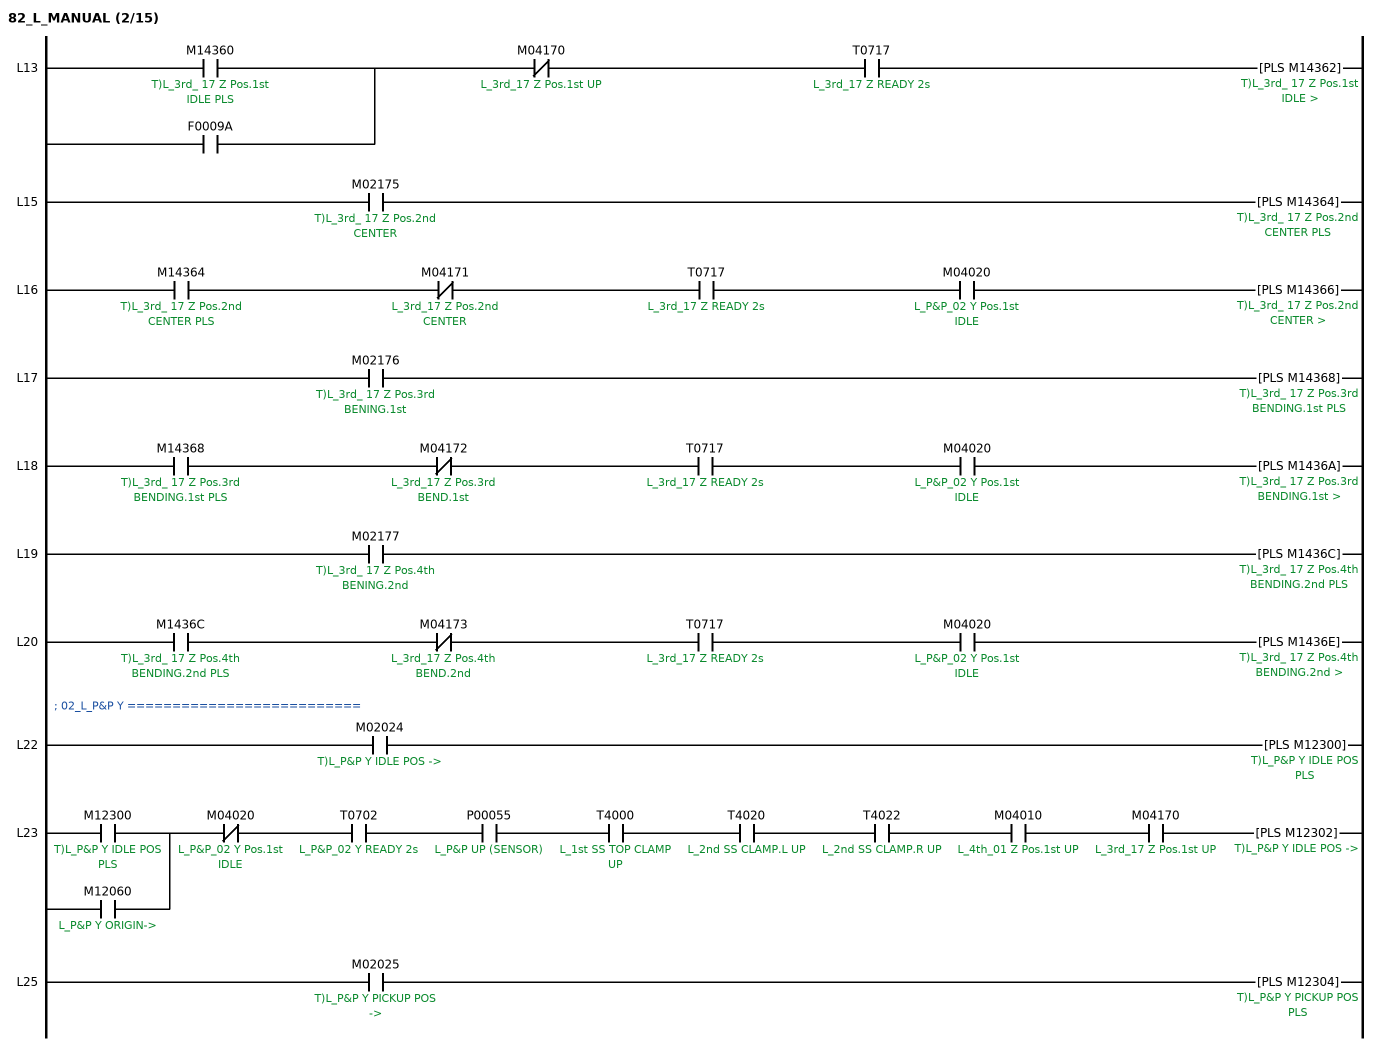
[picture p336: 82_L_MANUAL rungs L13-L25]
; L13
LOAD      M14360	// T)L_3rd_ 17 Z Pos.1st IDLE PLS
OR        F0009A
AND NOT   M04170	// L_3rd_17 Z Pos.1st UP
AND       T0717	// L_3rd_17 Z READY 2s
OUTP      M14362	// T)L_3rd_ 17 Z Pos.1st IDLE >
; L15
LOAD      M02175	// T)L_3rd_ 17 Z Pos.2nd CENTER
OUTP      M14364	// T)L_3rd_ 17 Z Pos.2nd CENTER PLS
; L16
LOAD      M14364	// T)L_3rd_ 17 Z Pos.2nd CENTER PLS
AND NOT   M04171	// L_3rd_17 Z Pos.2nd CENTER
AND       T0717	// L_3rd_17 Z READY 2s
AND       M04020	// L_P&P_02 Y Pos.1st IDLE
OUTP      M14366	// T)L_3rd_ 17 Z Pos.2nd CENTER >
; L17
LOAD      M02176	// T)L_3rd_ 17 Z Pos.3rd BENING.1st
OUTP      M14368	// T)L_3rd_ 17 Z Pos.3rd BENDING.1st PLS
; L18
LOAD      M14368	// T)L_3rd_ 17 Z Pos.3rd BENDING.1st PLS
AND NOT   M04172	// L_3rd_17 Z Pos.3rd BEND.1st
AND       T0717	// L_3rd_17 Z READY 2s
AND       M04020	// L_P&P_02 Y Pos.1st IDLE
OUTP      M1436A	// T)L_3rd_ 17 Z Pos.3rd BENDING.1st >
; L19
LOAD      M02177	// T)L_3rd_ 17 Z Pos.4th BENING.2nd
OUTP      M1436C	// T)L_3rd_ 17 Z Pos.4th BENDING.2nd PLS
; L20
LOAD      M1436C	// T)L_3rd_ 17 Z Pos.4th BENDING.2nd PLS
AND NOT   M04173	// L_3rd_17 Z Pos.4th BEND.2nd
AND       T0717	// L_3rd_17 Z READY 2s
AND       M04020	// L_P&P_02 Y Pos.1st IDLE
OUTP      M1436E	// T)L_3rd_ 17 Z Pos.4th BENDING.2nd >
// 02_L_P&P Y ==========================
; L22
LOAD      M02024	// T)L_P&P Y IDLE POS ->
OUTP      M12300	// T)L_P&P Y IDLE POS PLS
; L23
LOAD      M12300	// T)L_P&P Y IDLE POS PLS
OR        M12060	// L_P&P Y ORIGIN->
AND NOT   M04020	// L_P&P_02 Y Pos.1st IDLE
AND       T0702	// L_P&P_02 Y READY 2s
AND       P00055	// L_P&P UP (SENSOR)
AND       T4000	// L_1st SS TOP CLAMP    UP
AND       T4020	// L_2nd SS CLAMP.L UP
AND       T4022	// L_2nd SS CLAMP.R UP
AND       M04010	// L_4th_01 Z Pos.1st UP
AND       M04170	// L_3rd_17 Z Pos.1st UP
OUTP      M12302	// T)L_P&P Y IDLE POS ->
; L25
LOAD      M02025	// T)L_P&P Y PICKUP POS ->
OUTP      M12304	// T)L_P&P Y PICKUP POS PLS

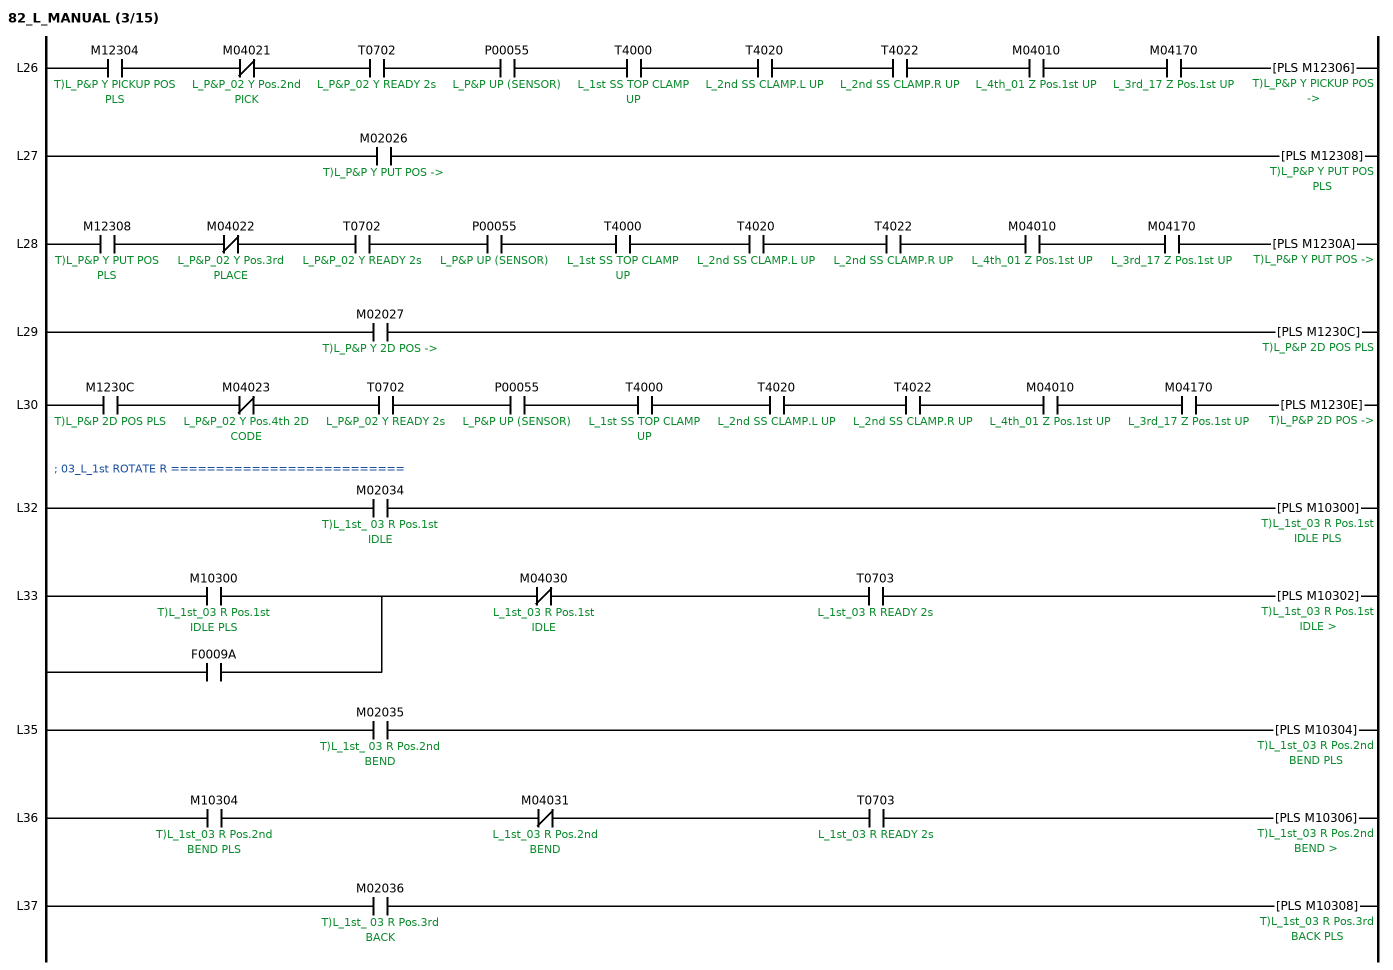
; L26
LOAD      M12304	// T)L_P&P Y PICKUP POS PLS
AND NOT   M04021	// L_P&P_02 Y Pos.2nd PICK
AND       T0702	// L_P&P_02 Y READY 2s
AND       P00055	// L_P&P UP (SENSOR)
AND       T4000	// L_1st SS TOP CLAMP    UP
AND       T4020	// L_2nd SS CLAMP.L UP
AND       T4022	// L_2nd SS CLAMP.R UP
AND       M04010	// L_4th_01 Z Pos.1st UP
AND       M04170	// L_3rd_17 Z Pos.1st UP
OUTP      M12306	// T)L_P&P Y PICKUP POS ->
; L27
LOAD      M02026	// T)L_P&P Y PUT POS ->
OUTP      M12308	// T)L_P&P Y PUT POS PLS
; L28
LOAD      M12308	// T)L_P&P Y PUT POS PLS
AND NOT   M04022	// L_P&P_02 Y Pos.3rd PLACE
AND       T0702	// L_P&P_02 Y READY 2s
AND       P00055	// L_P&P UP (SENSOR)
AND       T4000	// L_1st SS TOP CLAMP    UP
AND       T4020	// L_2nd SS CLAMP.L UP
AND       T4022	// L_2nd SS CLAMP.R UP
AND       M04010	// L_4th_01 Z Pos.1st UP
AND       M04170	// L_3rd_17 Z Pos.1st UP
OUTP      M1230A	// T)L_P&P Y PUT POS ->
; L29
LOAD      M02027	// T)L_P&P Y 2D POS ->
OUTP      M1230C	// T)L_P&P 2D POS PLS
; L30
LOAD      M1230C	// T)L_P&P 2D POS PLS
AND NOT   M04023	// L_P&P_02 Y Pos.4th 2D CODE
AND       T0702	// L_P&P_02 Y READY 2s
AND       P00055	// L_P&P UP (SENSOR)
AND       T4000	// L_1st SS TOP CLAMP    UP
AND       T4020	// L_2nd SS CLAMP.L UP
AND       T4022	// L_2nd SS CLAMP.R UP
AND       M04010	// L_4th_01 Z Pos.1st UP
AND       M04170	// L_3rd_17 Z Pos.1st UP
OUTP      M1230E	// T)L_P&P 2D POS ->
// 03_L_1st ROTATE R ==========================
; L32
LOAD      M02034	// T)L_1st_ 03 R Pos.1st IDLE
OUTP      M10300	// T)L_1st_03 R Pos.1st IDLE PLS
; L33
LOAD      M10300	// T)L_1st_03 R Pos.1st IDLE PLS
OR        F0009A
AND NOT   M04030	// L_1st_03 R Pos.1st IDLE
AND       T0703	// L_1st_03 R READY 2s
OUTP      M10302	// T)L_1st_03 R Pos.1st IDLE >
; L35
LOAD      M02035	// T)L_1st_ 03 R Pos.2nd BEND
OUTP      M10304	// T)L_1st_03 R Pos.2nd BEND PLS
; L36
LOAD      M10304	// T)L_1st_03 R Pos.2nd BEND PLS
AND NOT   M04031	// L_1st_03 R Pos.2nd BEND
AND       T0703	// L_1st_03 R READY 2s
OUTP      M10306	// T)L_1st_03 R Pos.2nd BEND >
; L37
LOAD      M02036	// T)L_1st_ 03 R Pos.3rd BACK
OUTP      M10308	// T)L_1st_03 R Pos.3rd BACK PLS

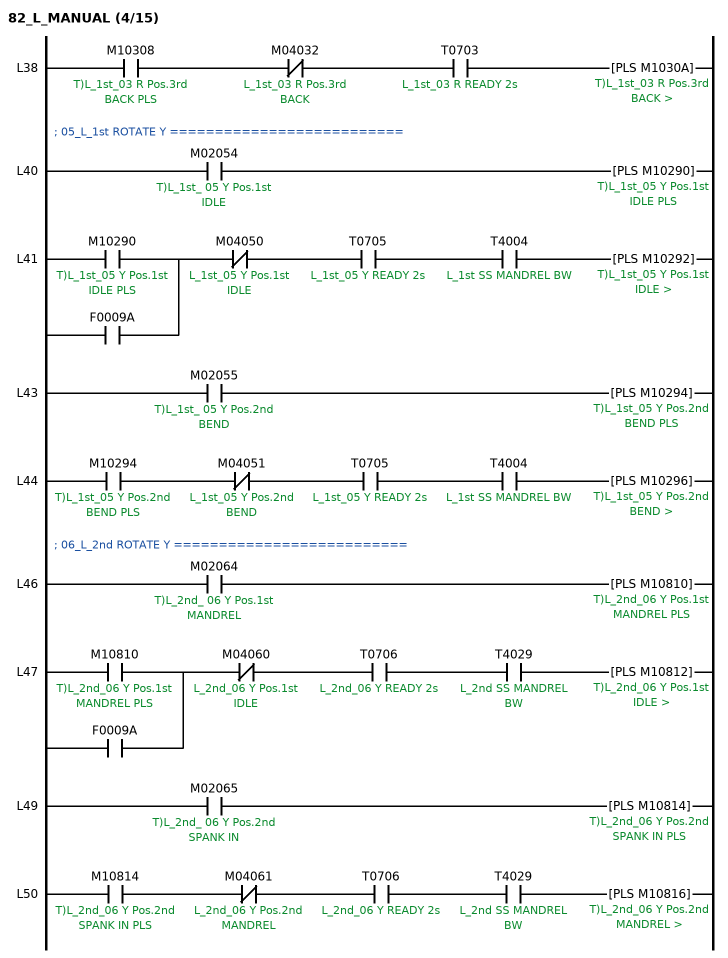
; L38
LOAD      M10308	// T)L_1st_03 R Pos.3rd BACK PLS
AND NOT   M04032	// L_1st_03 R Pos.3rd BACK
AND       T0703	// L_1st_03 R READY 2s
OUTP      M1030A	// T)L_1st_03 R Pos.3rd BACK >
// 05_L_1st ROTATE Y ==========================
; L40
LOAD      M02054	// T)L_1st_ 05 Y Pos.1st IDLE
OUTP      M10290	// T)L_1st_05 Y Pos.1st IDLE PLS
; L41
LOAD      M10290	// T)L_1st_05 Y Pos.1st IDLE PLS
OR        F0009A
AND NOT   M04050	// L_1st_05 Y Pos.1st IDLE
AND       T0705	// L_1st_05 Y READY 2s
AND       T4004	// L_1st SS MANDREL BW
OUTP      M10292	// T)L_1st_05 Y Pos.1st IDLE >
; L43
LOAD      M02055	// T)L_1st_ 05 Y Pos.2nd BEND
OUTP      M10294	// T)L_1st_05 Y Pos.2nd BEND PLS
; L44
LOAD      M10294	// T)L_1st_05 Y Pos.2nd BEND PLS
AND NOT   M04051	// L_1st_05 Y Pos.2nd BEND
AND       T0705	// L_1st_05 Y READY 2s
AND       T4004	// L_1st SS MANDREL BW
OUTP      M10296	// T)L_1st_05 Y Pos.2nd BEND >
// 06_L_2nd ROTATE Y ==========================
; L46
LOAD      M02064	// T)L_2nd_ 06 Y Pos.1st MANDREL
OUTP      M10810	// T)L_2nd_06 Y Pos.1st MANDREL PLS
; L47
LOAD      M10810	// T)L_2nd_06 Y Pos.1st MANDREL PLS
OR        F0009A
AND NOT   M04060	// L_2nd_06 Y Pos.1st IDLE
AND       T0706	// L_2nd_06 Y READY 2s
AND       T4029	// L_2nd SS MANDREL BW
OUTP      M10812	// T)L_2nd_06 Y Pos.1st IDLE >
; L49
LOAD      M02065	// T)L_2nd_ 06 Y Pos.2nd SPANK IN
OUTP      M10814	// T)L_2nd_06 Y Pos.2nd SPANK IN PLS
; L50
LOAD      M10814	// T)L_2nd_06 Y Pos.2nd SPANK IN PLS
AND NOT   M04061	// L_2nd_06 Y Pos.2nd MANDREL
AND       T0706	// L_2nd_06 Y READY 2s
AND       T4029	// L_2nd SS MANDREL BW
OUTP      M10816	// T)L_2nd_06 Y Pos.2nd MANDREL >

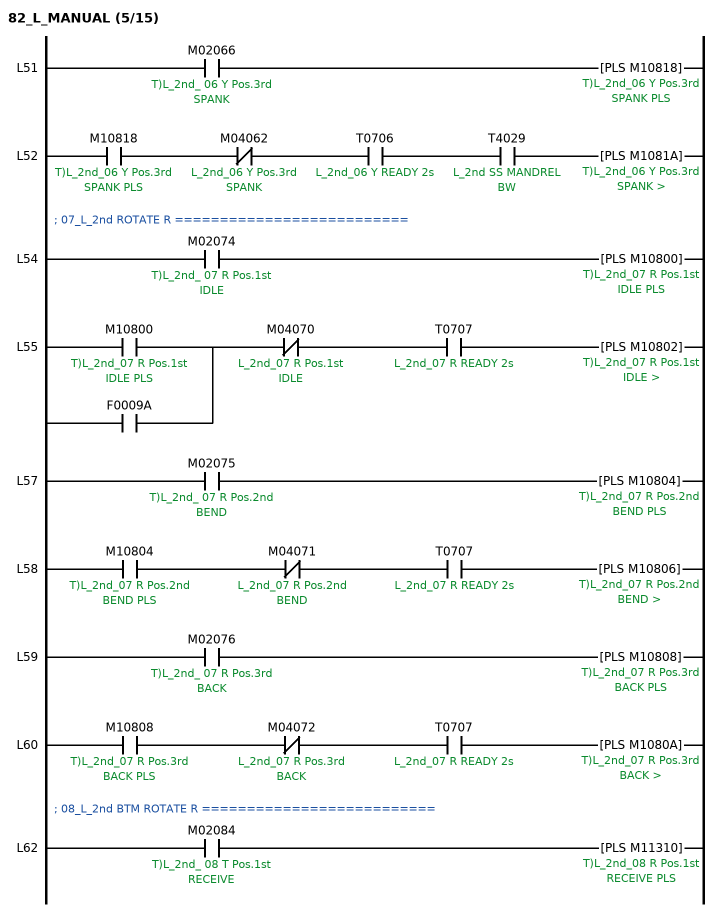
; L51
LOAD      M02066	// T)L_2nd_ 06 Y Pos.3rd SPANK
OUTP      M10818	// T)L_2nd_06 Y Pos.3rd SPANK PLS
; L52
LOAD      M10818	// T)L_2nd_06 Y Pos.3rd SPANK PLS
AND NOT   M04062	// L_2nd_06 Y Pos.3rd SPANK
AND       T0706	// L_2nd_06 Y READY 2s
AND       T4029	// L_2nd SS MANDREL BW
OUTP      M1081A	// T)L_2nd_06 Y Pos.3rd SPANK >
// 07_L_2nd ROTATE R ==========================
; L54
LOAD      M02074	// T)L_2nd_ 07 R Pos.1st IDLE
OUTP      M10800	// T)L_2nd_07 R Pos.1st IDLE PLS
; L55
LOAD      M10800	// T)L_2nd_07 R Pos.1st IDLE PLS
OR        F0009A
AND NOT   M04070	// L_2nd_07 R Pos.1st IDLE
AND       T0707	// L_2nd_07 R READY 2s
OUTP      M10802	// T)L_2nd_07 R Pos.1st IDLE >
; L57
LOAD      M02075	// T)L_2nd_ 07 R Pos.2nd BEND
OUTP      M10804	// T)L_2nd_07 R Pos.2nd BEND PLS
; L58
LOAD      M10804	// T)L_2nd_07 R Pos.2nd BEND PLS
AND NOT   M04071	// L_2nd_07 R Pos.2nd BEND
AND       T0707	// L_2nd_07 R READY 2s
OUTP      M10806	// T)L_2nd_07 R Pos.2nd BEND >
; L59
LOAD      M02076	// T)L_2nd_ 07 R Pos.3rd BACK
OUTP      M10808	// T)L_2nd_07 R Pos.3rd BACK PLS
; L60
LOAD      M10808	// T)L_2nd_07 R Pos.3rd BACK PLS
AND NOT   M04072	// L_2nd_07 R Pos.3rd BACK
AND       T0707	// L_2nd_07 R READY 2s
OUTP      M1080A	// T)L_2nd_07 R Pos.3rd BACK >
// 08_L_2nd BTM ROTATE R ==========================
; L62
LOAD      M02084	// T)L_2nd_ 08 T Pos.1st RECEIVE
OUTP      M11310	// T)L_2nd_08 R Pos.1st RECEIVE PLS

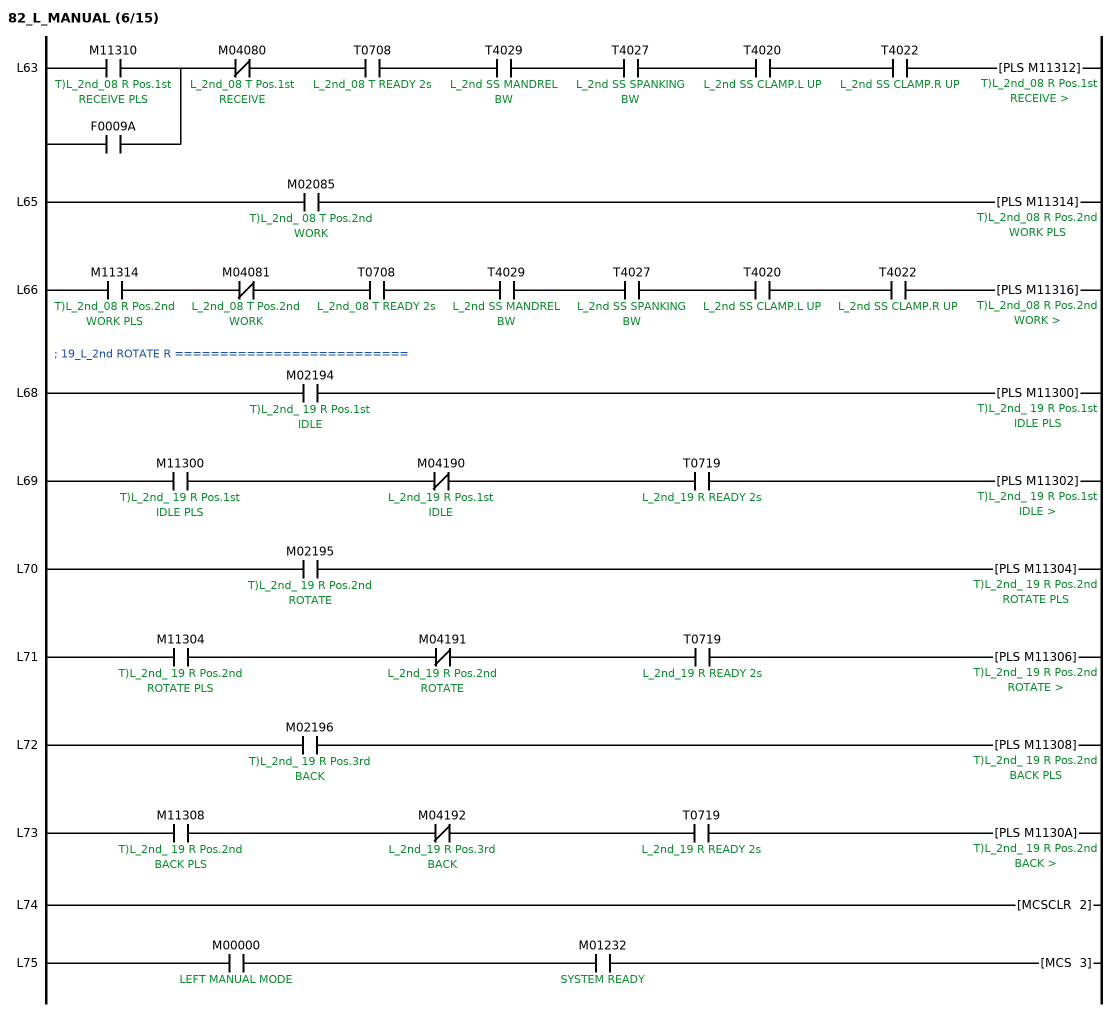
; L63
LOAD      M11310	// T)L_2nd_08 R Pos.1st RECEIVE PLS
OR        F0009A
AND NOT   M04080	// L_2nd_08 T Pos.1st RECEIVE
AND       T0708	// L_2nd_08 T READY 2s
AND       T4029	// L_2nd SS MANDREL BW
AND       T4027	// L_2nd SS SPANKING BW
AND       T4020	// L_2nd SS CLAMP.L UP
AND       T4022	// L_2nd SS CLAMP.R UP
OUTP      M11312	// T)L_2nd_08 R Pos.1st RECEIVE >
; L65
LOAD      M02085	// T)L_2nd_ 08 T Pos.2nd WORK
OUTP      M11314	// T)L_2nd_08 R Pos.2nd WORK PLS
; L66
LOAD      M11314	// T)L_2nd_08 R Pos.2nd WORK PLS
AND NOT   M04081	// L_2nd_08 T Pos.2nd WORK
AND       T0708	// L_2nd_08 T READY 2s
AND       T4029	// L_2nd SS MANDREL BW
AND       T4027	// L_2nd SS SPANKING BW
AND       T4020	// L_2nd SS CLAMP.L UP
AND       T4022	// L_2nd SS CLAMP.R UP
OUTP      M11316	// T)L_2nd_08 R Pos.2nd WORK >
// 19_L_2nd ROTATE R ==========================
; L68
LOAD      M02194	// T)L_2nd_ 19 R Pos.1st IDLE
OUTP      M11300	// T)L_2nd_ 19 R Pos.1st IDLE PLS
; L69
LOAD      M11300	// T)L_2nd_ 19 R Pos.1st IDLE PLS
AND NOT   M04190	// L_2nd_19 R Pos.1st IDLE
AND       T0719	// L_2nd_19 R READY 2s
OUTP      M11302	// T)L_2nd_ 19 R Pos.1st IDLE >
; L70
LOAD      M02195	// T)L_2nd_ 19 R Pos.2nd ROTATE
OUTP      M11304	// T)L_2nd_ 19 R Pos.2nd ROTATE PLS
; L71
LOAD      M11304	// T)L_2nd_ 19 R Pos.2nd ROTATE PLS
AND NOT   M04191	// L_2nd_19 R Pos.2nd ROTATE
AND       T0719	// L_2nd_19 R READY 2s
OUTP      M11306	// T)L_2nd_ 19 R Pos.2nd ROTATE >
; L72
LOAD      M02196	// T)L_2nd_ 19 R Pos.3rd BACK
OUTP      M11308	// T)L_2nd_ 19 R Pos.2nd BACK PLS
; L73
LOAD      M11308	// T)L_2nd_ 19 R Pos.2nd BACK PLS
AND NOT   M04192	// L_2nd_19 R Pos.3rd BACK
AND       T0719	// L_2nd_19 R READY 2s
OUTP      M1130A	// T)L_2nd_ 19 R Pos.2nd BACK >
; L74
MCSCLR    2
; L75
LOAD      M00000	// LEFT MANUAL MODE
AND       M01232	// SYSTEM READY
MCS       3

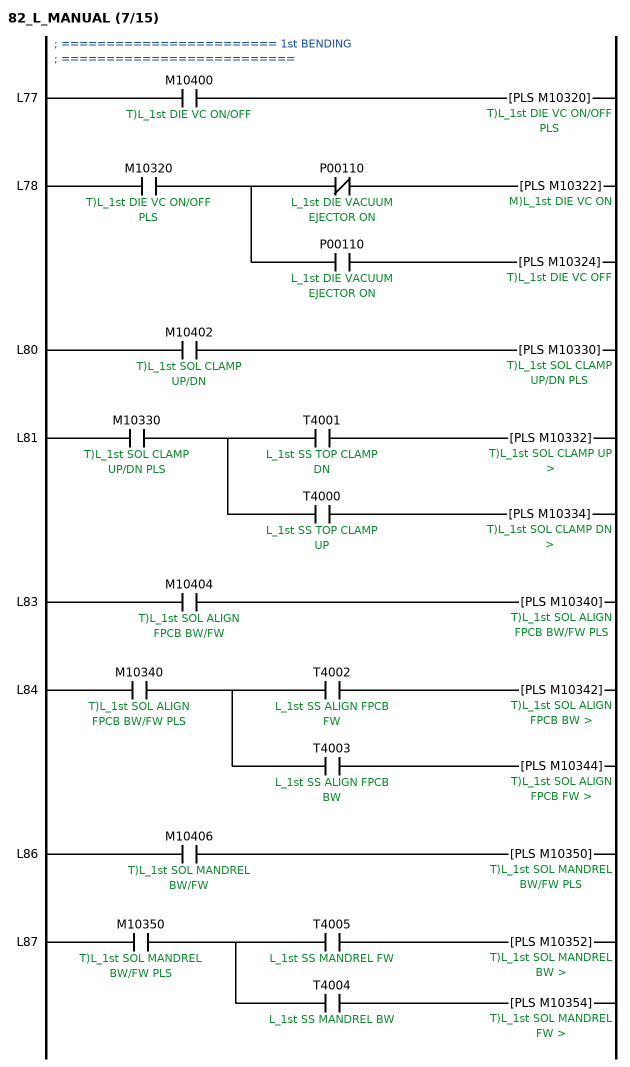
// ======================== 1st BENDING ==========================
; L77
LOAD      M10400	// T)L_1st DIE VC ON/OFF
OUTP      M10320	// T)L_1st DIE VC ON/OFF PLS
; L78
LOAD      M10320	// T)L_1st DIE VC ON/OFF PLS
MPUSH
AND NOT   P00110	// L_1st DIE VACUUM EJECTOR ON
OUTP      M10322	// M)L_1st DIE VC ON
MPOP
AND       P00110	// L_1st DIE VACUUM EJECTOR ON
OUTP      M10324	// T)L_1st DIE VC OFF
; L80
LOAD      M10402	// T)L_1st SOL CLAMP UP/DN
OUTP      M10330	// T)L_1st SOL CLAMP UP/DN PLS
; L81
LOAD      M10330	// T)L_1st SOL CLAMP UP/DN PLS
MPUSH
AND       T4001	// L_1st SS TOP CLAMP    DN
OUTP      M10332	// T)L_1st SOL CLAMP UP >
MPOP
AND       T4000	// L_1st SS TOP CLAMP    UP
OUTP      M10334	// T)L_1st SOL CLAMP DN >
; L83
LOAD      M10404	// T)L_1st SOL ALIGN FPCB BW/FW
OUTP      M10340	// T)L_1st SOL ALIGN FPCB BW/FW PLS
; L84
LOAD      M10340	// T)L_1st SOL ALIGN FPCB BW/FW PLS
MPUSH
AND       T4002	// L_1st SS ALIGN FPCB FW
OUTP      M10342	// T)L_1st SOL ALIGN FPCB BW >
MPOP
AND       T4003	// L_1st SS ALIGN FPCB BW
OUTP      M10344	// T)L_1st SOL ALIGN FPCB FW >
; L86
LOAD      M10406	// T)L_1st SOL MANDREL BW/FW
OUTP      M10350	// T)L_1st SOL MANDREL BW/FW PLS
; L87
LOAD      M10350	// T)L_1st SOL MANDREL BW/FW PLS
MPUSH
AND       T4005	// L_1st SS MANDREL FW
OUTP      M10352	// T)L_1st SOL MANDREL BW >
MPOP
AND       T4004	// L_1st SS MANDREL BW
OUTP      M10354	// T)L_1st SOL MANDREL FW >

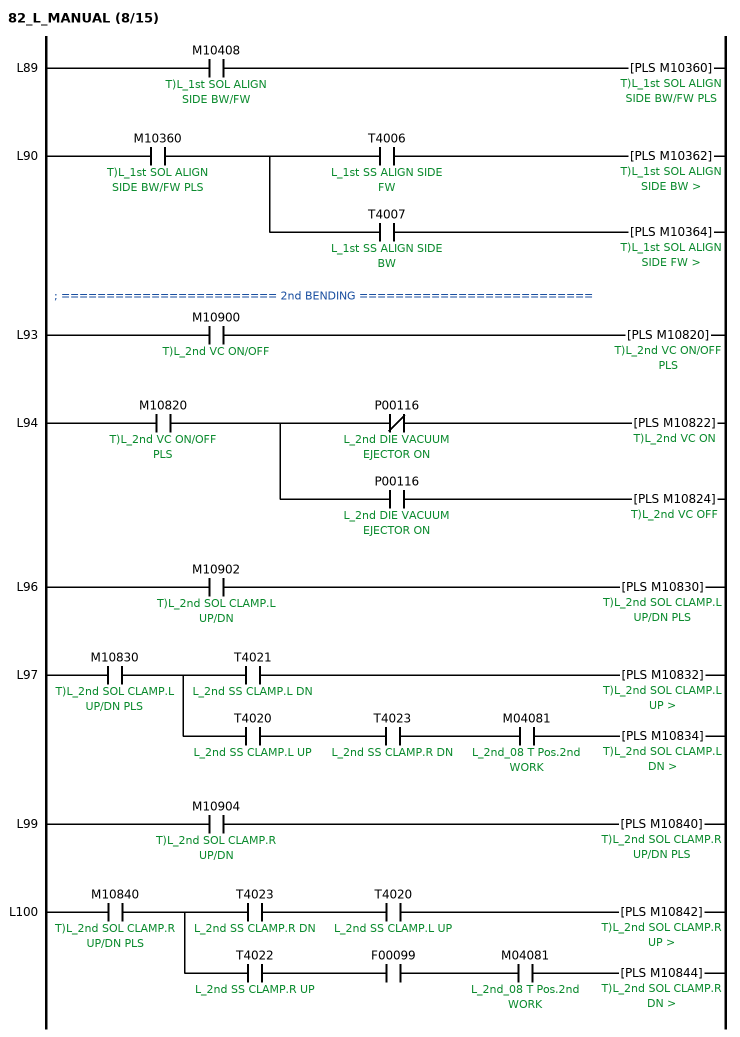
; L89
LOAD      M10408	// T)L_1st SOL ALIGN SIDE BW/FW
OUTP      M10360	// T)L_1st SOL ALIGN SIDE BW/FW PLS
; L90
LOAD      M10360	// T)L_1st SOL ALIGN SIDE BW/FW PLS
MPUSH
AND       T4006	// L_1st SS ALIGN SIDE FW
OUTP      M10362	// T)L_1st SOL ALIGN SIDE BW >
MPOP
AND       T4007	// L_1st SS ALIGN SIDE BW
OUTP      M10364	// T)L_1st SOL ALIGN SIDE FW >
// ======================== 2nd BENDING ==========================
; L93
LOAD      M10900	// T)L_2nd VC ON/OFF
OUTP      M10820	// T)L_2nd VC ON/OFF PLS
; L94
LOAD      M10820	// T)L_2nd VC ON/OFF PLS
MPUSH
AND NOT   P00116	// L_2nd DIE VACUUM EJECTOR ON
OUTP      M10822	// T)L_2nd VC ON
MPOP
AND       P00116	// L_2nd DIE VACUUM EJECTOR ON
OUTP      M10824	// T)L_2nd VC OFF
; L96
LOAD      M10902	// T)L_2nd SOL CLAMP.L UP/DN
OUTP      M10830	// T)L_2nd SOL CLAMP.L UP/DN PLS
; L97
LOAD      M10830	// T)L_2nd SOL CLAMP.L UP/DN PLS
MPUSH
AND       T4021	// L_2nd SS CLAMP.L DN
OUTP      M10832	// T)L_2nd SOL CLAMP.L UP >
MPOP
AND       T4020	// L_2nd SS CLAMP.L UP
AND       T4023	// L_2nd SS CLAMP.R DN
AND       M04081	// L_2nd_08 T Pos.2nd WORK
OUTP      M10834	// T)L_2nd SOL CLAMP.L DN >
; L99
LOAD      M10904	// T)L_2nd SOL CLAMP.R UP/DN
OUTP      M10840	// T)L_2nd SOL CLAMP.R UP/DN PLS
; L100
LOAD      M10840	// T)L_2nd SOL CLAMP.R UP/DN PLS
MPUSH
AND       T4023	// L_2nd SS CLAMP.R DN
AND       T4020	// L_2nd SS CLAMP.L UP
OUTP      M10842	// T)L_2nd SOL CLAMP.R UP >
MPOP
AND       T4022	// L_2nd SS CLAMP.R UP
AND       F00099
AND       M04081	// L_2nd_08 T Pos.2nd WORK
OUTP      M10844	// T)L_2nd SOL CLAMP.R DN >

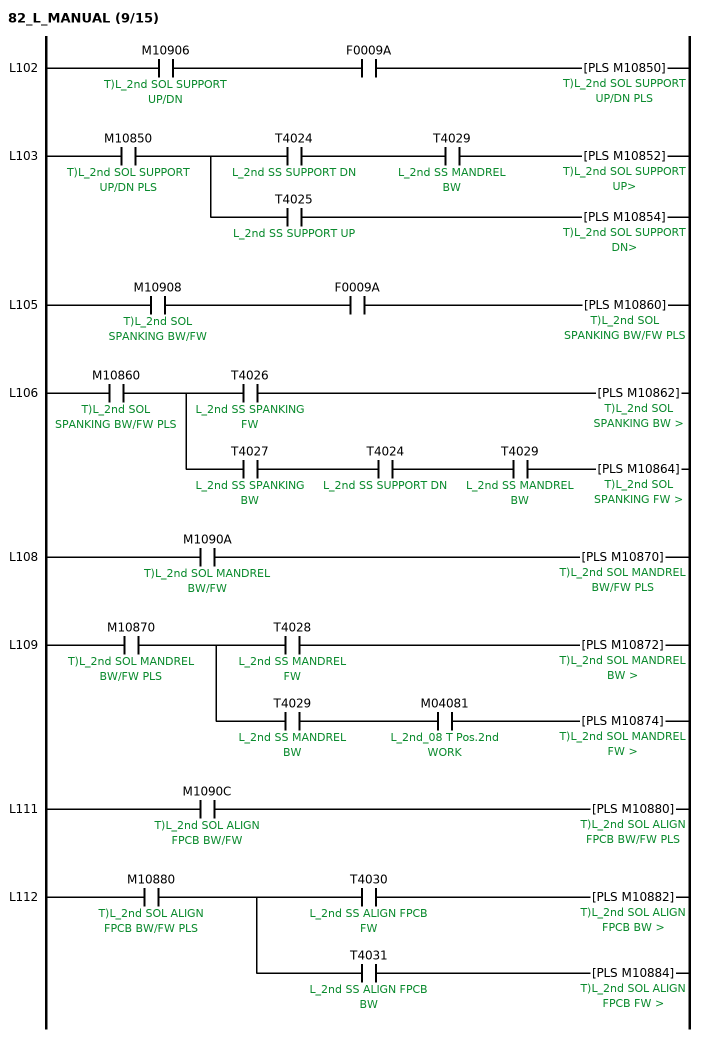
; L102
LOAD      M10906	// T)L_2nd SOL SUPPORT UP/DN
AND       F0009A
OUTP      M10850	// T)L_2nd SOL SUPPORT UP/DN PLS
; L103
LOAD      M10850	// T)L_2nd SOL SUPPORT UP/DN PLS
MPUSH
AND       T4024	// L_2nd SS SUPPORT DN
AND       T4029	// L_2nd SS MANDREL BW
OUTP      M10852	// T)L_2nd SOL SUPPORT UP>
MPOP
AND       T4025	// L_2nd SS SUPPORT UP
OUTP      M10854	// T)L_2nd SOL SUPPORT DN>
; L105
LOAD      M10908	// T)L_2nd SOL SPANKING BW/FW
AND       F0009A
OUTP      M10860	// T)L_2nd SOL SPANKING BW/FW PLS
; L106
LOAD      M10860	// T)L_2nd SOL SPANKING BW/FW PLS
MPUSH
AND       T4026	// L_2nd SS SPANKING FW
OUTP      M10862	// T)L_2nd SOL SPANKING BW >
MPOP
AND       T4027	// L_2nd SS SPANKING BW
AND       T4024	// L_2nd SS SUPPORT DN
AND       T4029	// L_2nd SS MANDREL BW
OUTP      M10864	// T)L_2nd SOL SPANKING FW >
; L108
LOAD      M1090A	// T)L_2nd SOL MANDREL BW/FW
OUTP      M10870	// T)L_2nd SOL MANDREL BW/FW PLS
; L109
LOAD      M10870	// T)L_2nd SOL MANDREL BW/FW PLS
MPUSH
AND       T4028	// L_2nd SS MANDREL FW
OUTP      M10872	// T)L_2nd SOL MANDREL BW >
MPOP
AND       T4029	// L_2nd SS MANDREL BW
AND       M04081	// L_2nd_08 T Pos.2nd WORK
OUTP      M10874	// T)L_2nd SOL MANDREL FW >
; L111
LOAD      M1090C	// T)L_2nd SOL ALIGN FPCB BW/FW
OUTP      M10880	// T)L_2nd SOL ALIGN FPCB BW/FW PLS
; L112
LOAD      M10880	// T)L_2nd SOL ALIGN FPCB BW/FW PLS
MPUSH
AND       T4030	// L_2nd SS ALIGN FPCB FW
OUTP      M10882	// T)L_2nd SOL ALIGN FPCB BW >
MPOP
AND       T4031	// L_2nd SS ALIGN FPCB BW
OUTP      M10884	// T)L_2nd SOL ALIGN FPCB FW >

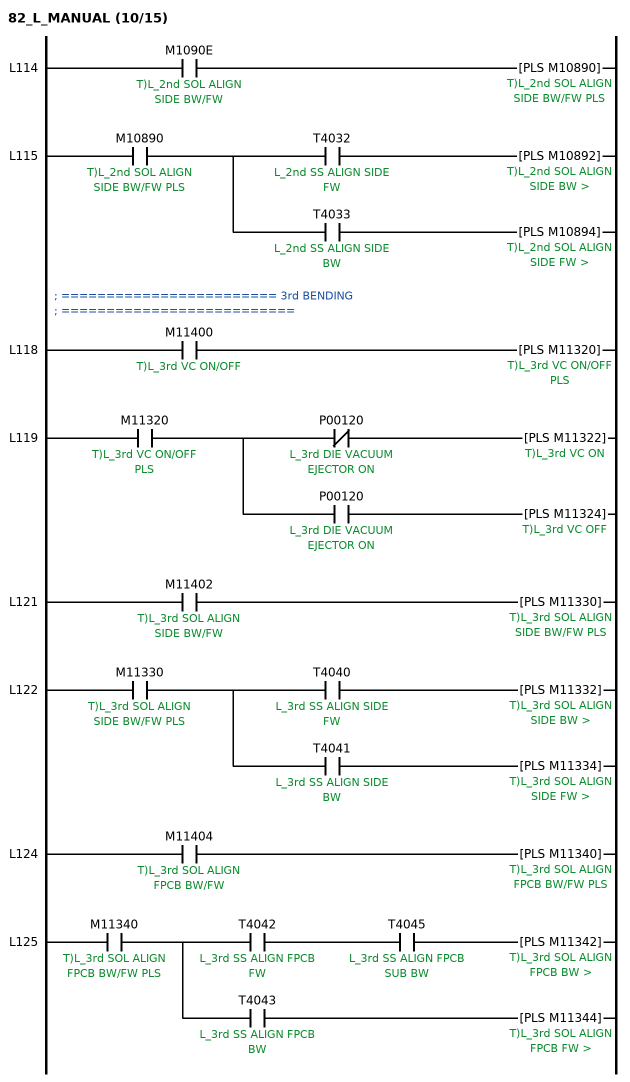
; L114
LOAD      M1090E	// T)L_2nd SOL ALIGN SIDE BW/FW
OUTP      M10890	// T)L_2nd SOL ALIGN SIDE BW/FW PLS
; L115
LOAD      M10890	// T)L_2nd SOL ALIGN SIDE BW/FW PLS
MPUSH
AND       T4032	// L_2nd SS ALIGN SIDE FW
OUTP      M10892	// T)L_2nd SOL ALIGN SIDE BW >
MPOP
AND       T4033	// L_2nd SS ALIGN SIDE BW
OUTP      M10894	// T)L_2nd SOL ALIGN SIDE FW >
// ======================== 3rd BENDING ==========================
; L118
LOAD      M11400	// T)L_3rd VC ON/OFF
OUTP      M11320	// T)L_3rd VC ON/OFF PLS
; L119
LOAD      M11320	// T)L_3rd VC ON/OFF PLS
MPUSH
AND NOT   P00120	// L_3rd DIE VACUUM EJECTOR ON
OUTP      M11322	// T)L_3rd VC ON
MPOP
AND       P00120	// L_3rd DIE VACUUM EJECTOR ON
OUTP      M11324	// T)L_3rd VC OFF
; L121
LOAD      M11402	// T)L_3rd SOL ALIGN SIDE BW/FW
OUTP      M11330	// T)L_3rd SOL ALIGN SIDE BW/FW PLS
; L122
LOAD      M11330	// T)L_3rd SOL ALIGN SIDE BW/FW PLS
MPUSH
AND       T4040	// L_3rd SS ALIGN SIDE FW
OUTP      M11332	// T)L_3rd SOL ALIGN SIDE BW >
MPOP
AND       T4041	// L_3rd SS ALIGN SIDE BW
OUTP      M11334	// T)L_3rd SOL ALIGN SIDE FW >
; L124
LOAD      M11404	// T)L_3rd SOL ALIGN FPCB BW/FW
OUTP      M11340	// T)L_3rd SOL ALIGN FPCB BW/FW PLS
; L125
LOAD      M11340	// T)L_3rd SOL ALIGN FPCB BW/FW PLS
MPUSH
AND       T4042	// L_3rd SS ALIGN FPCB FW
AND       T4045	// L_3rd SS ALIGN FPCB SUB BW
OUTP      M11342	// T)L_3rd SOL ALIGN FPCB BW >
MPOP
AND       T4043	// L_3rd SS ALIGN FPCB BW
OUTP      M11344	// T)L_3rd SOL ALIGN FPCB FW >

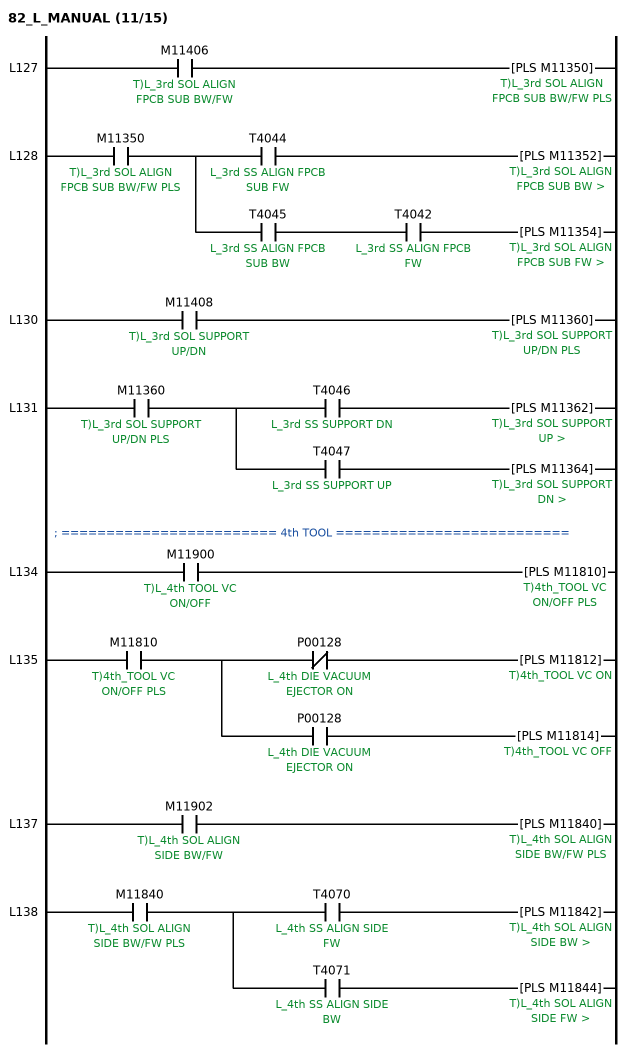
; L127
LOAD      M11406	// T)L_3rd SOL ALIGN FPCB SUB BW/FW
OUTP      M11350	// T)L_3rd SOL ALIGN FPCB SUB BW/FW PLS
; L128
LOAD      M11350	// T)L_3rd SOL ALIGN FPCB SUB BW/FW PLS
MPUSH
AND       T4044	// L_3rd SS ALIGN FPCB SUB FW
OUTP      M11352	// T)L_3rd SOL ALIGN FPCB SUB BW >
MPOP
AND       T4045	// L_3rd SS ALIGN FPCB SUB BW
AND       T4042	// L_3rd SS ALIGN FPCB FW
OUTP      M11354	// T)L_3rd SOL ALIGN FPCB SUB FW >
; L130
LOAD      M11408	// T)L_3rd SOL SUPPORT UP/DN
OUTP      M11360	// T)L_3rd SOL SUPPORT UP/DN PLS
; L131
LOAD      M11360	// T)L_3rd SOL SUPPORT UP/DN PLS
MPUSH
AND       T4046	// L_3rd SS SUPPORT DN
OUTP      M11362	// T)L_3rd SOL SUPPORT UP >
MPOP
AND       T4047	// L_3rd SS SUPPORT UP
OUTP      M11364	// T)L_3rd SOL SUPPORT DN >
// ======================== 4th TOOL ==========================
; L134
LOAD      M11900	// T)L_4th TOOL VC ON/OFF
OUTP      M11810	// T)4th_TOOL VC ON/OFF PLS
; L135
LOAD      M11810	// T)4th_TOOL VC ON/OFF PLS
MPUSH
AND NOT   P00128	// L_4th DIE VACUUM EJECTOR ON
OUTP      M11812	// T)4th_TOOL VC ON
MPOP
AND       P00128	// L_4th DIE VACUUM EJECTOR ON
OUTP      M11814	// T)4th_TOOL VC OFF
; L137
LOAD      M11902	// T)L_4th SOL ALIGN SIDE BW/FW
OUTP      M11840	// T)L_4th SOL ALIGN SIDE BW/FW PLS
; L138
LOAD      M11840	// T)L_4th SOL ALIGN SIDE BW/FW PLS
MPUSH
AND       T4070	// L_4th SS ALIGN SIDE FW
OUTP      M11842	// T)L_4th SOL ALIGN SIDE BW >
MPOP
AND       T4071	// L_4th SS ALIGN SIDE BW
OUTP      M11844	// T)L_4th SOL ALIGN SIDE FW >

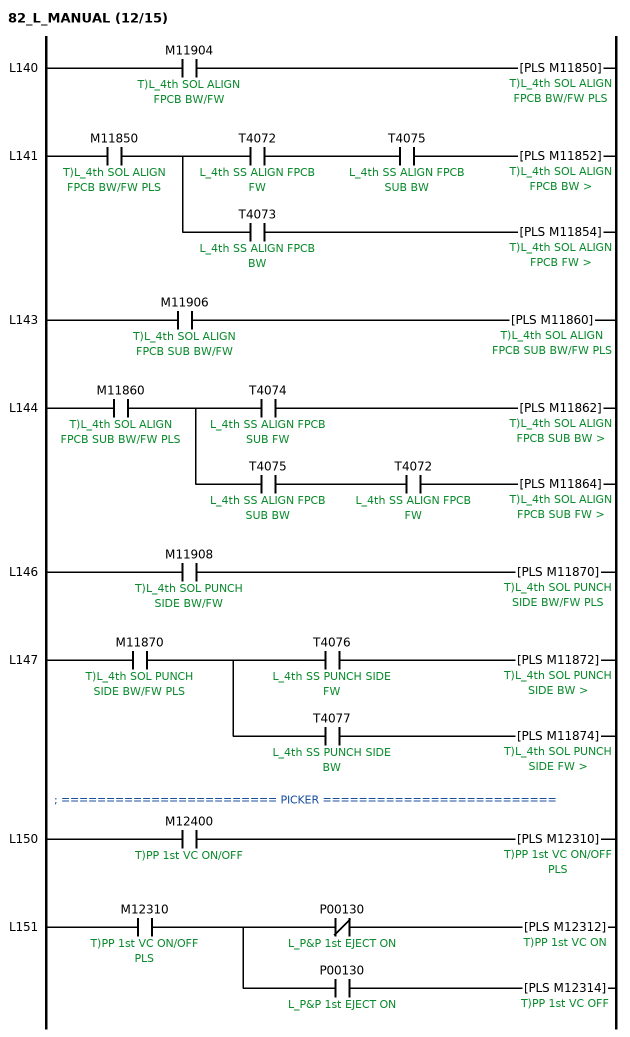
; L140
LOAD      M11904	// T)L_4th SOL ALIGN FPCB BW/FW
OUTP      M11850	// T)L_4th SOL ALIGN FPCB BW/FW PLS
; L141
LOAD      M11850	// T)L_4th SOL ALIGN FPCB BW/FW PLS
MPUSH
AND       T4072	// L_4th SS ALIGN FPCB FW
AND       T4075	// L_4th SS ALIGN FPCB SUB BW
OUTP      M11852	// T)L_4th SOL ALIGN FPCB BW >
MPOP
AND       T4073	// L_4th SS ALIGN FPCB BW
OUTP      M11854	// T)L_4th SOL ALIGN FPCB FW >
; L143
LOAD      M11906	// T)L_4th SOL ALIGN FPCB SUB BW/FW
OUTP      M11860	// T)L_4th SOL ALIGN FPCB SUB BW/FW PLS
; L144
LOAD      M11860	// T)L_4th SOL ALIGN FPCB SUB BW/FW PLS
MPUSH
AND       T4074	// L_4th SS ALIGN FPCB SUB FW
OUTP      M11862	// T)L_4th SOL ALIGN FPCB SUB BW >
MPOP
AND       T4075	// L_4th SS ALIGN FPCB SUB BW
AND       T4072	// L_4th SS ALIGN FPCB FW
OUTP      M11864	// T)L_4th SOL ALIGN FPCB SUB FW >
; L146
LOAD      M11908	// T)L_4th SOL PUNCH SIDE BW/FW
OUTP      M11870	// T)L_4th SOL PUNCH SIDE BW/FW PLS
; L147
LOAD      M11870	// T)L_4th SOL PUNCH SIDE BW/FW PLS
MPUSH
AND       T4076	// L_4th SS PUNCH SIDE FW
OUTP      M11872	// T)L_4th SOL PUNCH SIDE BW >
MPOP
AND       T4077	// L_4th SS PUNCH SIDE BW
OUTP      M11874	// T)L_4th SOL PUNCH SIDE FW >
// ======================== PICKER ==========================
; L150
LOAD      M12400	// T)PP 1st VC ON/OFF
OUTP      M12310	// T)PP 1st VC ON/OFF PLS
; L151
LOAD      M12310	// T)PP 1st VC ON/OFF PLS
MPUSH
AND NOT   P00130	// L_P&P 1st EJECT ON
OUTP      M12312	// T)PP 1st VC ON
MPOP
AND       P00130	// L_P&P 1st EJECT ON
OUTP      M12314	// T)PP 1st VC OFF

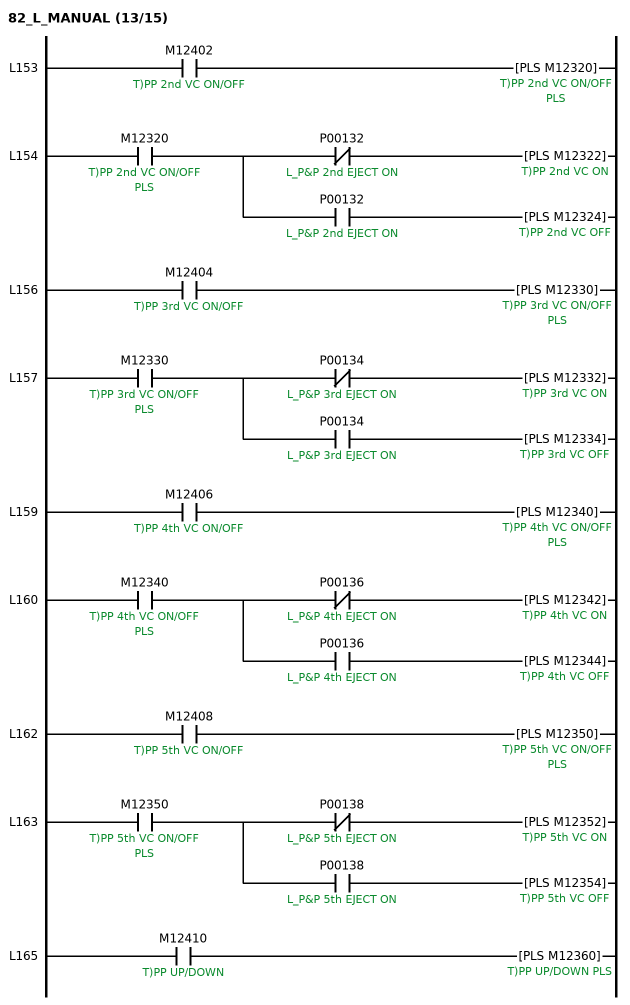
; L153
LOAD      M12402	// T)PP 2nd VC ON/OFF
OUTP      M12320	// T)PP 2nd VC ON/OFF PLS
; L154
LOAD      M12320	// T)PP 2nd VC ON/OFF PLS
MPUSH
AND NOT   P00132	// L_P&P 2nd EJECT ON
OUTP      M12322	// T)PP 2nd VC ON
MPOP
AND       P00132	// L_P&P 2nd EJECT ON
OUTP      M12324	// T)PP 2nd VC OFF
; L156
LOAD      M12404	// T)PP 3rd VC ON/OFF
OUTP      M12330	// T)PP 3rd VC ON/OFF PLS
; L157
LOAD      M12330	// T)PP 3rd VC ON/OFF PLS
MPUSH
AND NOT   P00134	// L_P&P 3rd EJECT ON
OUTP      M12332	// T)PP 3rd VC ON
MPOP
AND       P00134	// L_P&P 3rd EJECT ON
OUTP      M12334	// T)PP 3rd VC OFF
; L159
LOAD      M12406	// T)PP 4th VC ON/OFF
OUTP      M12340	// T)PP 4th VC ON/OFF PLS
; L160
LOAD      M12340	// T)PP 4th VC ON/OFF PLS
MPUSH
AND NOT   P00136	// L_P&P 4th EJECT ON
OUTP      M12342	// T)PP 4th VC ON
MPOP
AND       P00136	// L_P&P 4th EJECT ON
OUTP      M12344	// T)PP 4th VC OFF
; L162
LOAD      M12408	// T)PP 5th VC ON/OFF
OUTP      M12350	// T)PP 5th VC ON/OFF PLS
; L163
LOAD      M12350	// T)PP 5th VC ON/OFF PLS
MPUSH
AND NOT   P00138	// L_P&P 5th EJECT ON
OUTP      M12352	// T)PP 5th VC ON
MPOP
AND       P00138	// L_P&P 5th EJECT ON
OUTP      M12354	// T)PP 5th VC OFF
; L165
LOAD      M12410	// T)PP UP/DOWN
OUTP      M12360	// T)PP UP/DOWN PLS

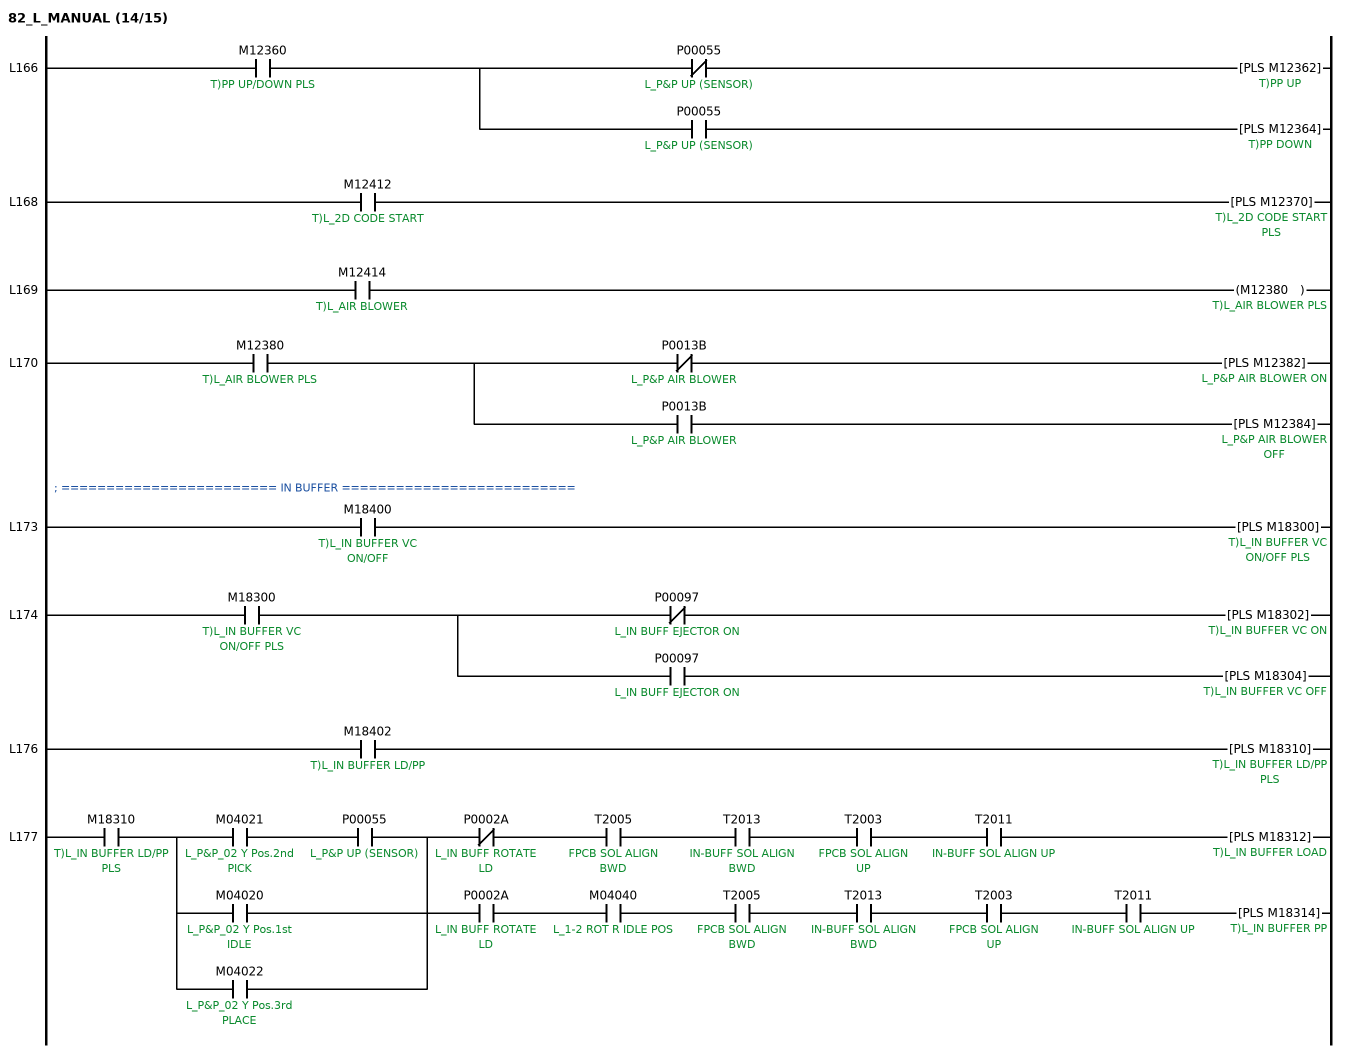
; L166
LOAD      M12360	// T)PP UP/DOWN PLS
MPUSH
AND NOT   P00055	// L_P&P UP (SENSOR)
OUTP      M12362	// T)PP UP
MPOP
AND       P00055	// L_P&P UP (SENSOR)
OUTP      M12364	// T)PP DOWN
; L168
LOAD      M12412	// T)L_2D CODE START
OUTP      M12370	// T)L_2D CODE START PLS
; L169
LOAD      M12414	// T)L_AIR BLOWER
OUT       M12380	// T)L_AIR BLOWER PLS
; L170
LOAD      M12380	// T)L_AIR BLOWER PLS
MPUSH
AND NOT   P0013B	// L_P&P AIR BLOWER
OUTP      M12382	// L_P&P AIR BLOWER ON
MPOP
AND       P0013B	// L_P&P AIR BLOWER
OUTP      M12384	// L_P&P AIR BLOWER OFF
// ======================== IN BUFFER ==========================
; L173
LOAD      M18400	// T)L_IN BUFFER VC ON/OFF
OUTP      M18300	// T)L_IN BUFFER VC ON/OFF PLS
; L174
LOAD      M18300	// T)L_IN BUFFER VC ON/OFF PLS
MPUSH
AND NOT   P00097	// L_IN BUFF EJECTOR ON
OUTP      M18302	// T)L_IN BUFFER VC ON
MPOP
AND       P00097	// L_IN BUFF EJECTOR ON
OUTP      M18304	// T)L_IN BUFFER VC OFF
; L176
LOAD      M18402	// T)L_IN BUFFER LD/PP
OUTP      M18310	// T)L_IN BUFFER LD/PP PLS
; L177
LOAD      M18310	// T)L_IN BUFFER LD/PP PLS
LOAD      M04021	// L_P&P_02 Y Pos.2nd PICK
AND       P00055	// L_P&P UP (SENSOR)
OR        M04020	// L_P&P_02 Y Pos.1st IDLE
OR        M04022	// L_P&P_02 Y Pos.3rd PLACE
AND LOAD
MPUSH
AND NOT   P0002A	// L_IN BUFF ROTATE     LD
AND       T2005	// FPCB SOL ALIGN         BWD
AND       T2013	// IN-BUFF SOL ALIGN BWD
AND       T2003	// FPCB SOL ALIGN         UP
AND       T2011	// IN-BUFF SOL ALIGN UP
OUTP      M18312	// T)L_IN BUFFER LOAD
MPOP
AND       P0002A	// L_IN BUFF ROTATE     LD
AND       M04040	// L_1-2 ROT R IDLE POS
AND       T2005	// FPCB SOL ALIGN         BWD
AND       T2013	// IN-BUFF SOL ALIGN BWD
AND       T2003	// FPCB SOL ALIGN         UP
AND       T2011	// IN-BUFF SOL ALIGN UP
OUTP      M18314	// T)L_IN BUFFER PP

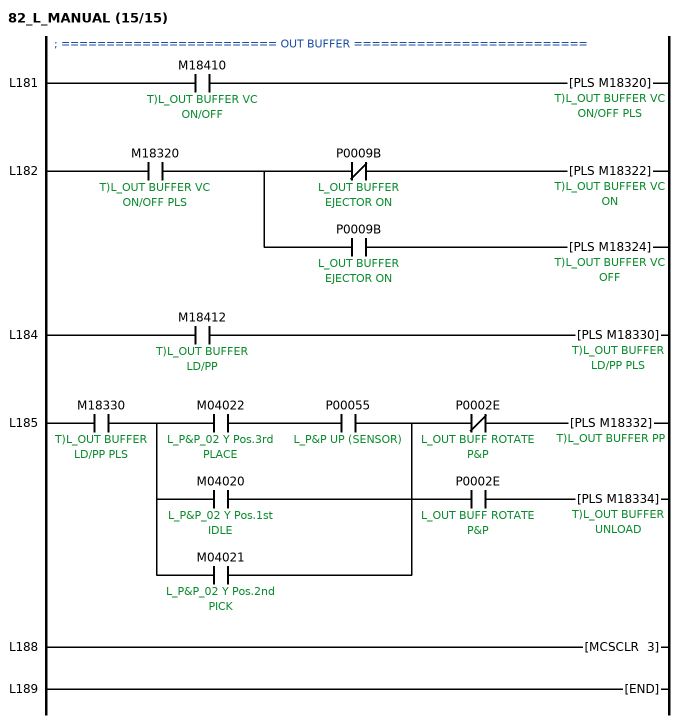
// ======================== OUT BUFFER ==========================
; L181
LOAD      M18410	// T)L_OUT BUFFER VC ON/OFF
OUTP      M18320	// T)L_OUT BUFFER VC ON/OFF PLS
; L182
LOAD      M18320	// T)L_OUT BUFFER VC ON/OFF PLS
MPUSH
AND NOT   P0009B	// L_OUT BUFFER EJECTOR ON
OUTP      M18322	// T)L_OUT BUFFER VC ON
MPOP
AND       P0009B	// L_OUT BUFFER EJECTOR ON
OUTP      M18324	// T)L_OUT BUFFER VC OFF
; L184
LOAD      M18412	// T)L_OUT BUFFER LD/PP
OUTP      M18330	// T)L_OUT BUFFER LD/PP PLS
; L185
LOAD      M18330	// T)L_OUT BUFFER LD/PP PLS
LOAD      M04022	// L_P&P_02 Y Pos.3rd PLACE
AND       P00055	// L_P&P UP (SENSOR)
OR        M04020	// L_P&P_02 Y Pos.1st IDLE
OR        M04021	// L_P&P_02 Y Pos.2nd PICK
AND LOAD
MPUSH
AND NOT   P0002E	// L_OUT BUFF ROTATE      P&P
OUTP      M18332	// T)L_OUT BUFFER PP
MPOP
AND       P0002E	// L_OUT BUFF ROTATE      P&P
OUTP      M18334	// T)L_OUT BUFFER UNLOAD
; L188
MCSCLR    3
; L189
END

PROGRAM 83_R_MANUAL (task: ¨ö¨¬A¥ì CA¡¤I¡¾¡¿¡¤¡Í)

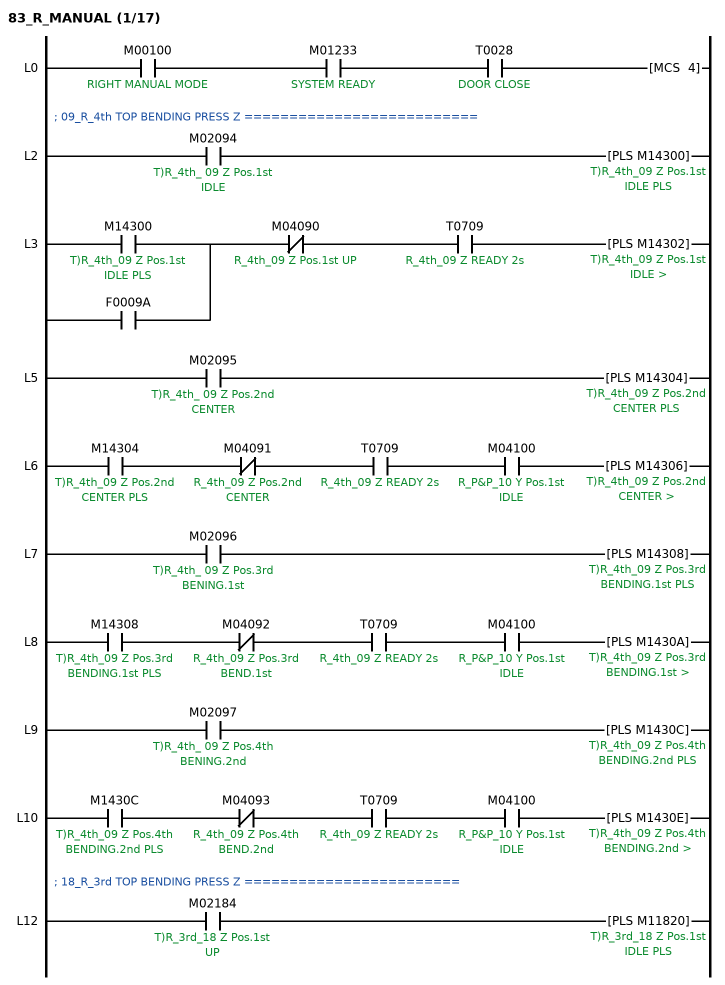
; L0
LOAD      M00100	// RIGHT MANUAL MODE
AND       M01233	// SYSTEM READY
AND       T0028	// DOOR CLOSE
MCS       4
// 09_R_4th TOP BENDING PRESS Z ==========================
; L2
LOAD      M02094	// T)R_4th_ 09 Z Pos.1st IDLE
OUTP      M14300	// T)R_4th_09 Z Pos.1st IDLE PLS
; L3
LOAD      M14300	// T)R_4th_09 Z Pos.1st IDLE PLS
OR        F0009A
AND NOT   M04090	// R_4th_09 Z Pos.1st UP
AND       T0709	// R_4th_09 Z READY 2s
OUTP      M14302	// T)R_4th_09 Z Pos.1st IDLE >
; L5
LOAD      M02095	// T)R_4th_ 09 Z Pos.2nd CENTER
OUTP      M14304	// T)R_4th_09 Z Pos.2nd CENTER PLS
; L6
LOAD      M14304	// T)R_4th_09 Z Pos.2nd CENTER PLS
AND NOT   M04091	// R_4th_09 Z Pos.2nd CENTER
AND       T0709	// R_4th_09 Z READY 2s
AND       M04100	// R_P&P_10 Y Pos.1st IDLE
OUTP      M14306	// T)R_4th_09 Z Pos.2nd CENTER >
; L7
LOAD      M02096	// T)R_4th_ 09 Z Pos.3rd BENING.1st
OUTP      M14308	// T)R_4th_09 Z Pos.3rd BENDING.1st PLS
; L8
LOAD      M14308	// T)R_4th_09 Z Pos.3rd BENDING.1st PLS
AND NOT   M04092	// R_4th_09 Z Pos.3rd BEND.1st
AND       T0709	// R_4th_09 Z READY 2s
AND       M04100	// R_P&P_10 Y Pos.1st IDLE
OUTP      M1430A	// T)R_4th_09 Z Pos.3rd BENDING.1st >
; L9
LOAD      M02097	// T)R_4th_ 09 Z Pos.4th BENING.2nd
OUTP      M1430C	// T)R_4th_09 Z Pos.4th BENDING.2nd PLS
; L10
LOAD      M1430C	// T)R_4th_09 Z Pos.4th BENDING.2nd PLS
AND NOT   M04093	// R_4th_09 Z Pos.4th BEND.2nd
AND       T0709	// R_4th_09 Z READY 2s
AND       M04100	// R_P&P_10 Y Pos.1st IDLE
OUTP      M1430E	// T)R_4th_09 Z Pos.4th BENDING.2nd >
// 18_R_3rd TOP BENDING PRESS Z ======================== 
; L12
LOAD      M02184	// T)R_3rd_18 Z Pos.1st UP
OUTP      M11820	// T)R_3rd_18 Z Pos.1st IDLE PLS

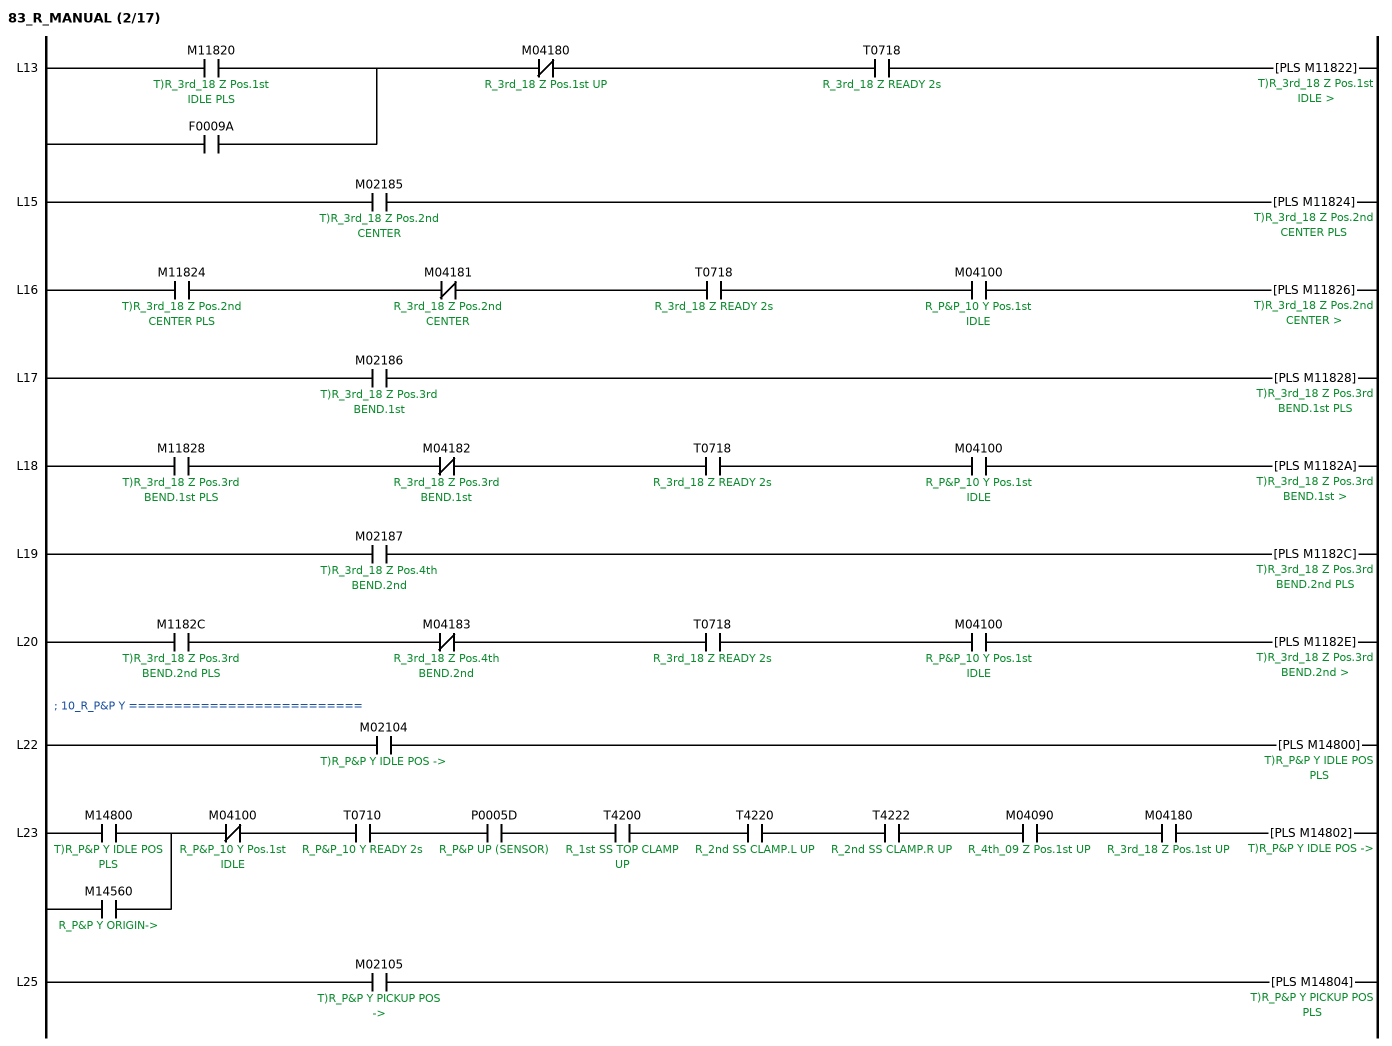
; L13
LOAD      M11820	// T)R_3rd_18 Z Pos.1st IDLE PLS
OR        F0009A
AND NOT   M04180	// R_3rd_18 Z Pos.1st UP
AND       T0718	// R_3rd_18 Z READY 2s
OUTP      M11822	// T)R_3rd_18 Z Pos.1st IDLE >
; L15
LOAD      M02185	// T)R_3rd_18 Z Pos.2nd CENTER
OUTP      M11824	// T)R_3rd_18 Z Pos.2nd CENTER PLS
; L16
LOAD      M11824	// T)R_3rd_18 Z Pos.2nd CENTER PLS
AND NOT   M04181	// R_3rd_18 Z Pos.2nd CENTER
AND       T0718	// R_3rd_18 Z READY 2s
AND       M04100	// R_P&P_10 Y Pos.1st IDLE
OUTP      M11826	// T)R_3rd_18 Z Pos.2nd CENTER >
; L17
LOAD      M02186	// T)R_3rd_18 Z Pos.3rd BEND.1st
OUTP      M11828	// T)R_3rd_18 Z Pos.3rd BEND.1st PLS
; L18
LOAD      M11828	// T)R_3rd_18 Z Pos.3rd BEND.1st PLS
AND NOT   M04182	// R_3rd_18 Z Pos.3rd BEND.1st
AND       T0718	// R_3rd_18 Z READY 2s
AND       M04100	// R_P&P_10 Y Pos.1st IDLE
OUTP      M1182A	// T)R_3rd_18 Z Pos.3rd BEND.1st >
; L19
LOAD      M02187	// T)R_3rd_18 Z Pos.4th BEND.2nd
OUTP      M1182C	// T)R_3rd_18 Z Pos.3rd BEND.2nd PLS
; L20
LOAD      M1182C	// T)R_3rd_18 Z Pos.3rd BEND.2nd PLS
AND NOT   M04183	// R_3rd_18 Z Pos.4th BEND.2nd
AND       T0718	// R_3rd_18 Z READY 2s
AND       M04100	// R_P&P_10 Y Pos.1st IDLE
OUTP      M1182E	// T)R_3rd_18 Z Pos.3rd BEND.2nd >
// 10_R_P&P Y ==========================
; L22
LOAD      M02104	// T)R_P&P Y IDLE POS ->
OUTP      M14800	// T)R_P&P Y IDLE POS PLS
; L23
LOAD      M14800	// T)R_P&P Y IDLE POS PLS
OR        M14560	// R_P&P Y ORIGIN->
AND NOT   M04100	// R_P&P_10 Y Pos.1st IDLE
AND       T0710	// R_P&P_10 Y READY 2s
AND       P0005D	// R_P&P UP (SENSOR)
AND       T4200	// R_1st SS TOP CLAMP UP
AND       T4220	// R_2nd SS CLAMP.L UP
AND       T4222	// R_2nd SS CLAMP.R UP
AND       M04090	// R_4th_09 Z Pos.1st UP
AND       M04180	// R_3rd_18 Z Pos.1st UP
OUTP      M14802	// T)R_P&P Y IDLE POS ->
; L25
LOAD      M02105	// T)R_P&P Y PICKUP POS ->
OUTP      M14804	// T)R_P&P Y PICKUP POS PLS

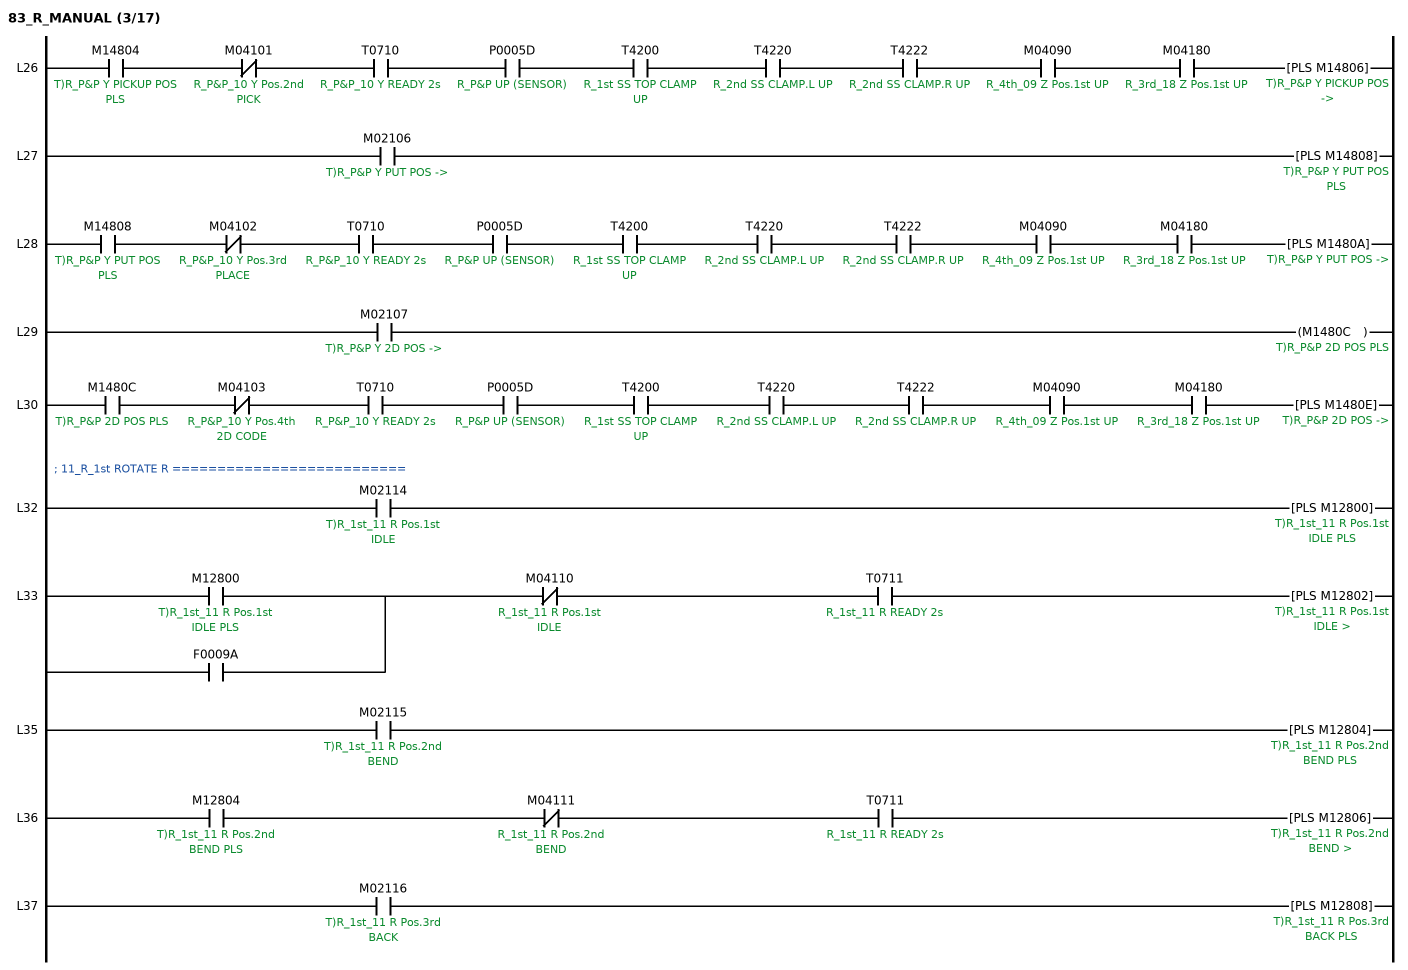
; L26
LOAD      M14804	// T)R_P&P Y PICKUP POS PLS
AND NOT   M04101	// R_P&P_10 Y Pos.2nd PICK
AND       T0710	// R_P&P_10 Y READY 2s
AND       P0005D	// R_P&P UP (SENSOR)
AND       T4200	// R_1st SS TOP CLAMP UP
AND       T4220	// R_2nd SS CLAMP.L UP
AND       T4222	// R_2nd SS CLAMP.R UP
AND       M04090	// R_4th_09 Z Pos.1st UP
AND       M04180	// R_3rd_18 Z Pos.1st UP
OUTP      M14806	// T)R_P&P Y PICKUP POS ->
; L27
LOAD      M02106	// T)R_P&P Y PUT POS ->
OUTP      M14808	// T)R_P&P Y PUT POS PLS
; L28
LOAD      M14808	// T)R_P&P Y PUT POS PLS
AND NOT   M04102	// R_P&P_10 Y Pos.3rd PLACE
AND       T0710	// R_P&P_10 Y READY 2s
AND       P0005D	// R_P&P UP (SENSOR)
AND       T4200	// R_1st SS TOP CLAMP UP
AND       T4220	// R_2nd SS CLAMP.L UP
AND       T4222	// R_2nd SS CLAMP.R UP
AND       M04090	// R_4th_09 Z Pos.1st UP
AND       M04180	// R_3rd_18 Z Pos.1st UP
OUTP      M1480A	// T)R_P&P Y PUT POS ->
; L29
LOAD      M02107	// T)R_P&P Y 2D POS ->
OUT       M1480C	// T)R_P&P 2D POS PLS
; L30
LOAD      M1480C	// T)R_P&P 2D POS PLS
AND NOT   M04103	// R_P&P_10 Y Pos.4th 2D CODE
AND       T0710	// R_P&P_10 Y READY 2s
AND       P0005D	// R_P&P UP (SENSOR)
AND       T4200	// R_1st SS TOP CLAMP UP
AND       T4220	// R_2nd SS CLAMP.L UP
AND       T4222	// R_2nd SS CLAMP.R UP
AND       M04090	// R_4th_09 Z Pos.1st UP
AND       M04180	// R_3rd_18 Z Pos.1st UP
OUTP      M1480E	// T)R_P&P 2D POS ->
// 11_R_1st ROTATE R ==========================
; L32
LOAD      M02114	// T)R_1st_11 R Pos.1st IDLE
OUTP      M12800	// T)R_1st_11 R Pos.1st IDLE PLS
; L33
LOAD      M12800	// T)R_1st_11 R Pos.1st IDLE PLS
OR        F0009A
AND NOT   M04110	// R_1st_11 R Pos.1st IDLE
AND       T0711	// R_1st_11 R READY 2s
OUTP      M12802	// T)R_1st_11 R Pos.1st IDLE >
; L35
LOAD      M02115	// T)R_1st_11 R Pos.2nd BEND
OUTP      M12804	// T)R_1st_11 R Pos.2nd BEND PLS
; L36
LOAD      M12804	// T)R_1st_11 R Pos.2nd BEND PLS
AND NOT   M04111	// R_1st_11 R Pos.2nd BEND
AND       T0711	// R_1st_11 R READY 2s
OUTP      M12806	// T)R_1st_11 R Pos.2nd BEND >
; L37
LOAD      M02116	// T)R_1st_11 R Pos.3rd BACK
OUTP      M12808	// T)R_1st_11 R Pos.3rd BACK PLS

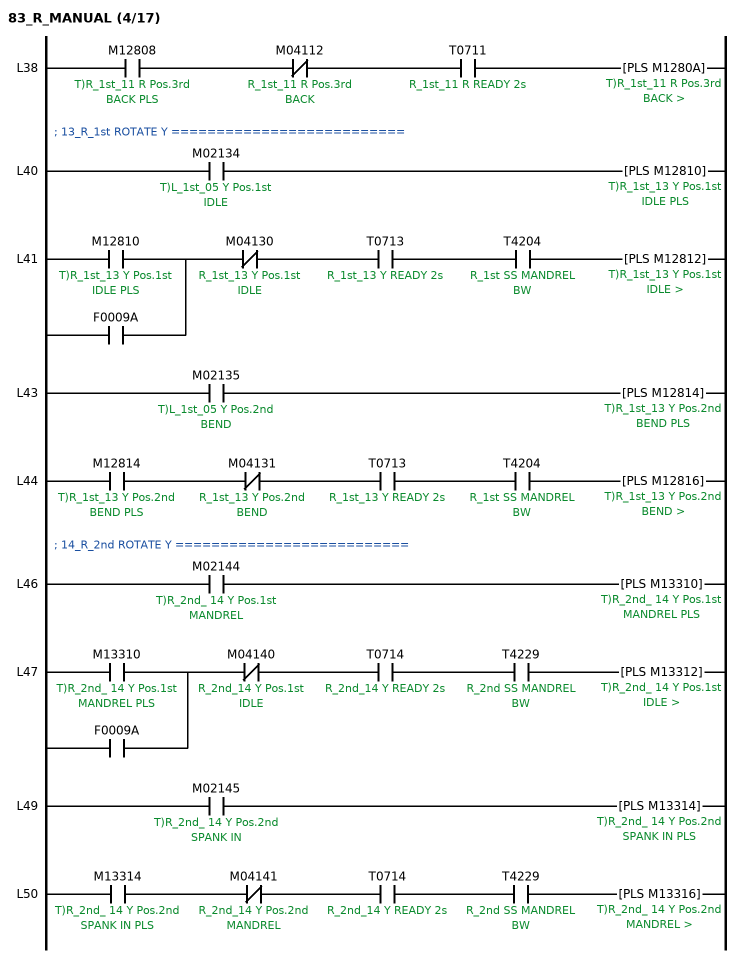
; L38
LOAD      M12808	// T)R_1st_11 R Pos.3rd BACK PLS
AND NOT   M04112	// R_1st_11 R Pos.3rd BACK
AND       T0711	// R_1st_11 R READY 2s
OUTP      M1280A	// T)R_1st_11 R Pos.3rd BACK >
// 13_R_1st ROTATE Y ==========================
; L40
LOAD      M02134	// T)L_1st_05 Y Pos.1st IDLE
OUTP      M12810	// T)R_1st_13 Y Pos.1st IDLE PLS
; L41
LOAD      M12810	// T)R_1st_13 Y Pos.1st IDLE PLS
OR        F0009A
AND NOT   M04130	// R_1st_13 Y Pos.1st IDLE
AND       T0713	// R_1st_13 Y READY 2s
AND       T4204	// R_1st SS MANDREL BW
OUTP      M12812	// T)R_1st_13 Y Pos.1st IDLE >
; L43
LOAD      M02135	// T)L_1st_05 Y Pos.2nd BEND
OUTP      M12814	// T)R_1st_13 Y Pos.2nd BEND PLS
; L44
LOAD      M12814	// T)R_1st_13 Y Pos.2nd BEND PLS
AND NOT   M04131	// R_1st_13 Y Pos.2nd BEND
AND       T0713	// R_1st_13 Y READY 2s
AND       T4204	// R_1st SS MANDREL BW
OUTP      M12816	// T)R_1st_13 Y Pos.2nd BEND >
// 14_R_2nd ROTATE Y ==========================
; L46
LOAD      M02144	// T)R_2nd_ 14 Y Pos.1st MANDREL
OUTP      M13310	// T)R_2nd_ 14 Y Pos.1st MANDREL PLS
; L47
LOAD      M13310	// T)R_2nd_ 14 Y Pos.1st MANDREL PLS
OR        F0009A
AND NOT   M04140	// R_2nd_14 Y Pos.1st IDLE
AND       T0714	// R_2nd_14 Y READY 2s
AND       T4229	// R_2nd SS MANDREL BW
OUTP      M13312	// T)R_2nd_ 14 Y Pos.1st IDLE >
; L49
LOAD      M02145	// T)R_2nd_ 14 Y Pos.2nd SPANK IN
OUTP      M13314	// T)R_2nd_ 14 Y Pos.2nd SPANK IN PLS
; L50
LOAD      M13314	// T)R_2nd_ 14 Y Pos.2nd SPANK IN PLS
AND NOT   M04141	// R_2nd_14 Y Pos.2nd MANDREL
AND       T0714	// R_2nd_14 Y READY 2s
AND       T4229	// R_2nd SS MANDREL BW
OUTP      M13316	// T)R_2nd_ 14 Y Pos.2nd MANDREL >

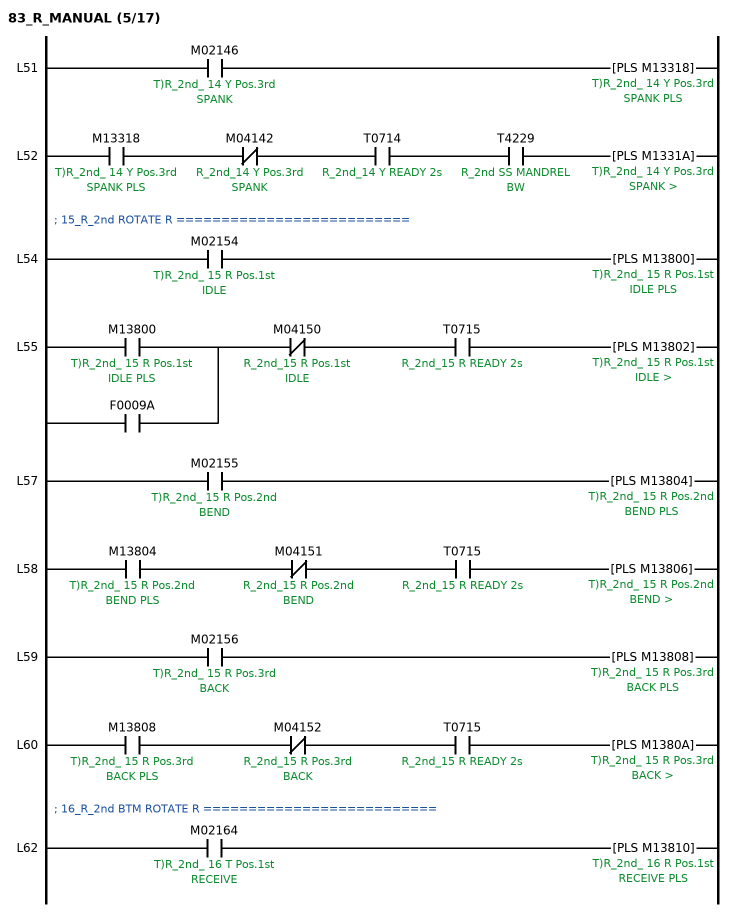
; L51
LOAD      M02146	// T)R_2nd_ 14 Y Pos.3rd SPANK
OUTP      M13318	// T)R_2nd_ 14 Y Pos.3rd SPANK PLS
; L52
LOAD      M13318	// T)R_2nd_ 14 Y Pos.3rd SPANK PLS
AND NOT   M04142	// R_2nd_14 Y Pos.3rd SPANK
AND       T0714	// R_2nd_14 Y READY 2s
AND       T4229	// R_2nd SS MANDREL BW
OUTP      M1331A	// T)R_2nd_ 14 Y Pos.3rd SPANK >
// 15_R_2nd ROTATE R ==========================
; L54
LOAD      M02154	// T)R_2nd_ 15 R Pos.1st IDLE
OUTP      M13800	// T)R_2nd_ 15 R Pos.1st IDLE PLS
; L55
LOAD      M13800	// T)R_2nd_ 15 R Pos.1st IDLE PLS
OR        F0009A
AND NOT   M04150	// R_2nd_15 R Pos.1st IDLE
AND       T0715	// R_2nd_15 R READY 2s
OUTP      M13802	// T)R_2nd_ 15 R Pos.1st IDLE >
; L57
LOAD      M02155	// T)R_2nd_ 15 R Pos.2nd BEND
OUTP      M13804	// T)R_2nd_ 15 R Pos.2nd BEND PLS
; L58
LOAD      M13804	// T)R_2nd_ 15 R Pos.2nd BEND PLS
AND NOT   M04151	// R_2nd_15 R Pos.2nd BEND
AND       T0715	// R_2nd_15 R READY 2s
OUTP      M13806	// T)R_2nd_ 15 R Pos.2nd BEND >
; L59
LOAD      M02156	// T)R_2nd_ 15 R Pos.3rd BACK
OUTP      M13808	// T)R_2nd_ 15 R Pos.3rd BACK PLS
; L60
LOAD      M13808	// T)R_2nd_ 15 R Pos.3rd BACK PLS
AND NOT   M04152	// R_2nd_15 R Pos.3rd BACK
AND       T0715	// R_2nd_15 R READY 2s
OUTP      M1380A	// T)R_2nd_ 15 R Pos.3rd BACK >
// 16_R_2nd BTM ROTATE R ==========================
; L62
LOAD      M02164	// T)R_2nd_ 16 T Pos.1st RECEIVE
OUTP      M13810	// T)R_2nd_ 16 R Pos.1st RECEIVE PLS

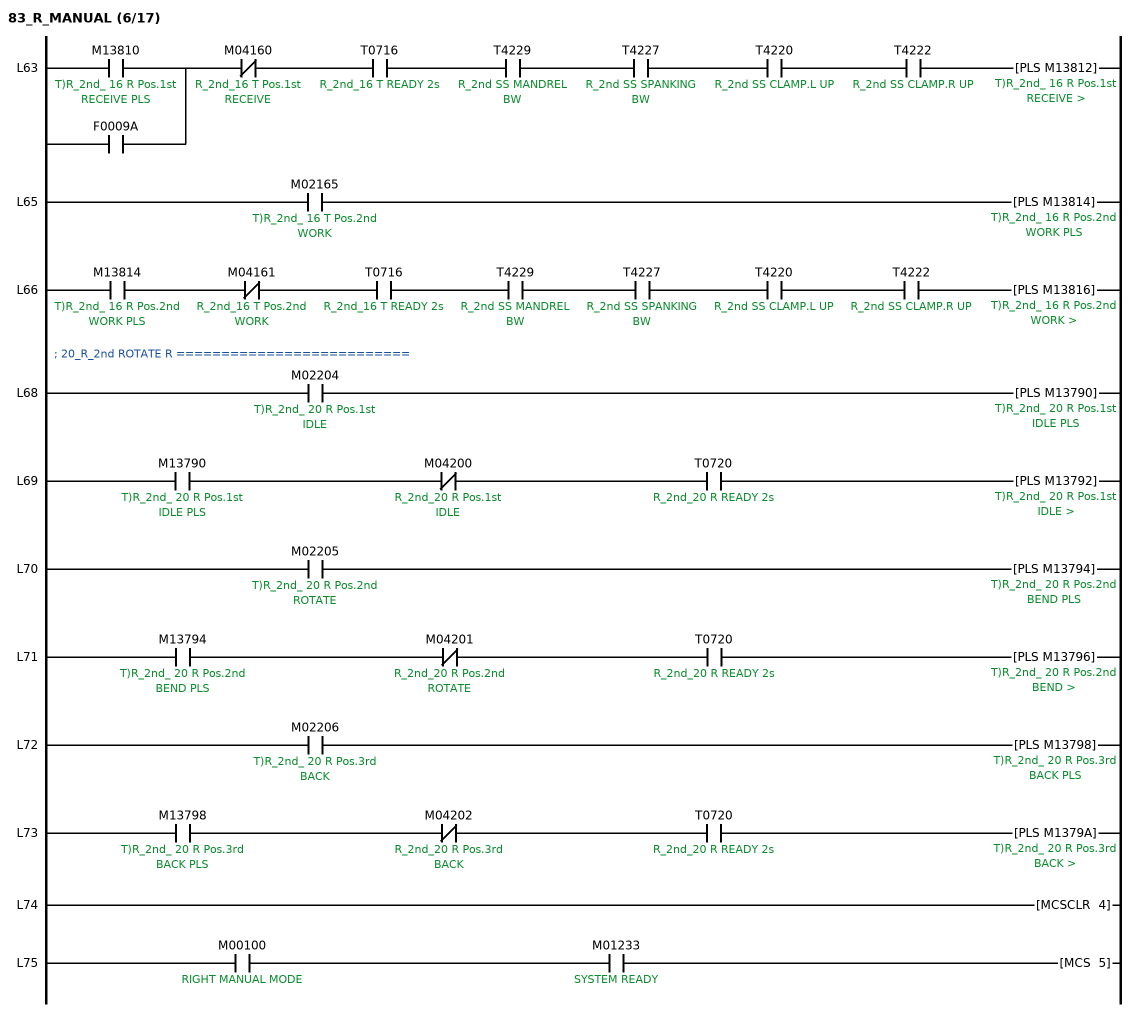
; L63
LOAD      M13810	// T)R_2nd_ 16 R Pos.1st RECEIVE PLS
OR        F0009A
AND NOT   M04160	// R_2nd_16 T Pos.1st RECEIVE
AND       T0716	// R_2nd_16 T READY 2s
AND       T4229	// R_2nd SS MANDREL BW
AND       T4227	// R_2nd SS SPANKING BW
AND       T4220	// R_2nd SS CLAMP.L UP
AND       T4222	// R_2nd SS CLAMP.R UP
OUTP      M13812	// T)R_2nd_ 16 R Pos.1st RECEIVE >
; L65
LOAD      M02165	// T)R_2nd_ 16 T Pos.2nd WORK
OUTP      M13814	// T)R_2nd_ 16 R Pos.2nd WORK PLS
; L66
LOAD      M13814	// T)R_2nd_ 16 R Pos.2nd WORK PLS
AND NOT   M04161	// R_2nd_16 T Pos.2nd WORK
AND       T0716	// R_2nd_16 T READY 2s
AND       T4229	// R_2nd SS MANDREL BW
AND       T4227	// R_2nd SS SPANKING BW
AND       T4220	// R_2nd SS CLAMP.L UP
AND       T4222	// R_2nd SS CLAMP.R UP
OUTP      M13816	// T)R_2nd_ 16 R Pos.2nd WORK >
// 20_R_2nd ROTATE R ==========================
; L68
LOAD      M02204	// T)R_2nd_ 20 R Pos.1st IDLE
OUTP      M13790	// T)R_2nd_ 20 R Pos.1st IDLE PLS
; L69
LOAD      M13790	// T)R_2nd_ 20 R Pos.1st IDLE PLS
AND NOT   M04200	// R_2nd_20 R Pos.1st IDLE
AND       T0720	// R_2nd_20 R READY 2s
OUTP      M13792	// T)R_2nd_ 20 R Pos.1st IDLE >
; L70
LOAD      M02205	// T)R_2nd_ 20 R Pos.2nd ROTATE
OUTP      M13794	// T)R_2nd_ 20 R Pos.2nd BEND PLS
; L71
LOAD      M13794	// T)R_2nd_ 20 R Pos.2nd BEND PLS
AND NOT   M04201	// R_2nd_20 R Pos.2nd ROTATE
AND       T0720	// R_2nd_20 R READY 2s
OUTP      M13796	// T)R_2nd_ 20 R Pos.2nd BEND >
; L72
LOAD      M02206	// T)R_2nd_ 20 R Pos.3rd BACK
OUTP      M13798	// T)R_2nd_ 20 R Pos.3rd BACK PLS
; L73
LOAD      M13798	// T)R_2nd_ 20 R Pos.3rd BACK PLS
AND NOT   M04202	// R_2nd_20 R Pos.3rd BACK
AND       T0720	// R_2nd_20 R READY 2s
OUTP      M1379A	// T)R_2nd_ 20 R Pos.3rd BACK >
; L74
MCSCLR    4
; L75
LOAD      M00100	// RIGHT MANUAL MODE
AND       M01233	// SYSTEM READY
MCS       5

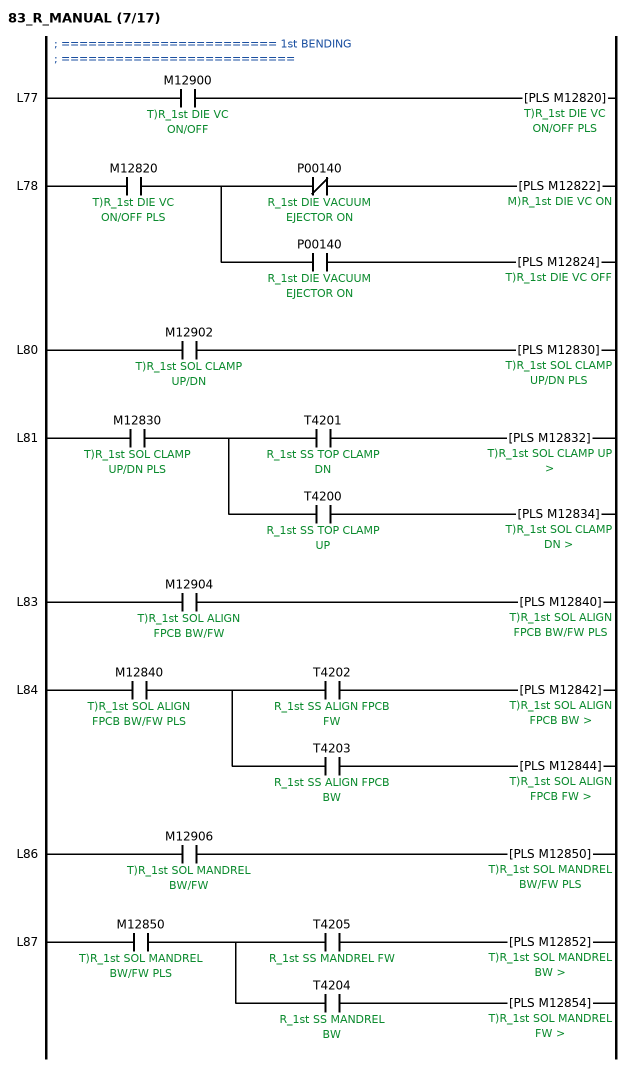
// ======================== 1st BENDING ==========================
; L77
LOAD      M12900	// T)R_1st DIE VC ON/OFF
OUTP      M12820	// T)R_1st DIE VC ON/OFF PLS
; L78
LOAD      M12820	// T)R_1st DIE VC ON/OFF PLS
MPUSH
AND NOT   P00140	// R_1st DIE VACUUM EJECTOR ON
OUTP      M12822	// M)R_1st DIE VC ON
MPOP
AND       P00140	// R_1st DIE VACUUM EJECTOR ON
OUTP      M12824	// T)R_1st DIE VC OFF
; L80
LOAD      M12902	// T)R_1st SOL CLAMP UP/DN
OUTP      M12830	// T)R_1st SOL CLAMP UP/DN PLS
; L81
LOAD      M12830	// T)R_1st SOL CLAMP UP/DN PLS
MPUSH
AND       T4201	// R_1st SS TOP CLAMP DN
OUTP      M12832	// T)R_1st SOL CLAMP UP >
MPOP
AND       T4200	// R_1st SS TOP CLAMP UP
OUTP      M12834	// T)R_1st SOL CLAMP DN >
; L83
LOAD      M12904	// T)R_1st SOL ALIGN FPCB BW/FW
OUTP      M12840	// T)R_1st SOL ALIGN FPCB BW/FW PLS
; L84
LOAD      M12840	// T)R_1st SOL ALIGN FPCB BW/FW PLS
MPUSH
AND       T4202	// R_1st SS ALIGN FPCB FW
OUTP      M12842	// T)R_1st SOL ALIGN FPCB BW >
MPOP
AND       T4203	// R_1st SS ALIGN FPCB BW
OUTP      M12844	// T)R_1st SOL ALIGN FPCB FW >
; L86
LOAD      M12906	// T)R_1st SOL MANDREL BW/FW
OUTP      M12850	// T)R_1st SOL MANDREL BW/FW PLS
; L87
LOAD      M12850	// T)R_1st SOL MANDREL BW/FW PLS
MPUSH
AND       T4205	// R_1st SS MANDREL FW
OUTP      M12852	// T)R_1st SOL MANDREL BW >
MPOP
AND       T4204	// R_1st SS MANDREL BW
OUTP      M12854	// T)R_1st SOL MANDREL FW >

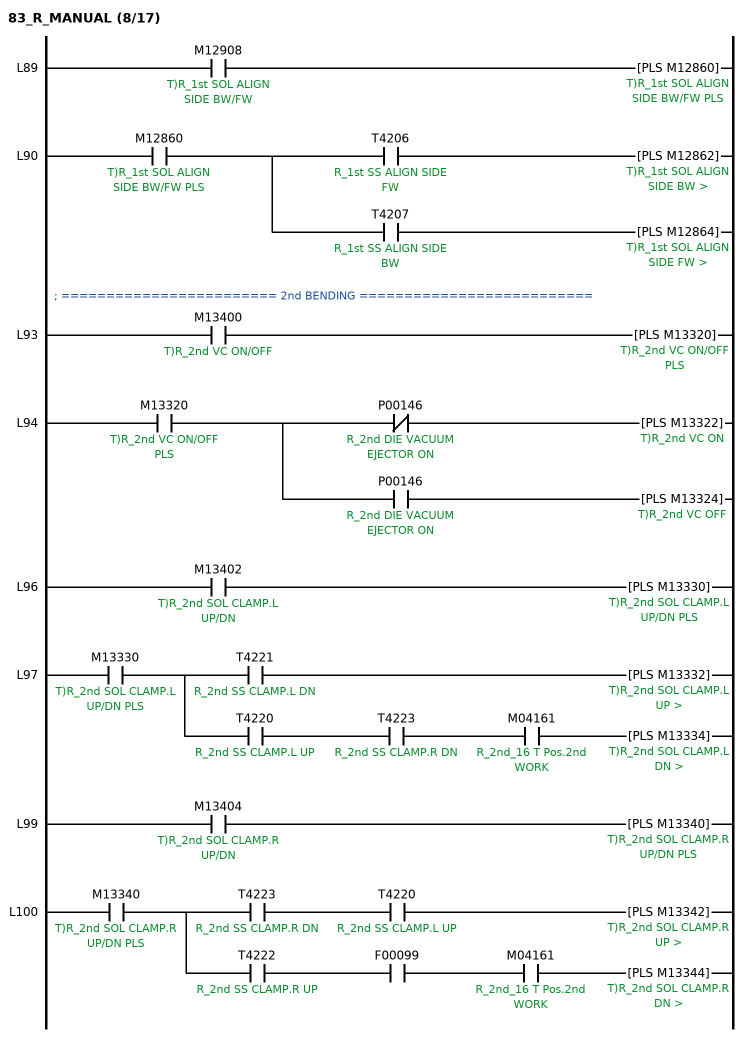
; L89
LOAD      M12908	// T)R_1st SOL ALIGN SIDE BW/FW
OUTP      M12860	// T)R_1st SOL ALIGN SIDE BW/FW PLS
; L90
LOAD      M12860	// T)R_1st SOL ALIGN SIDE BW/FW PLS
MPUSH
AND       T4206	// R_1st SS ALIGN SIDE FW
OUTP      M12862	// T)R_1st SOL ALIGN SIDE BW >
MPOP
AND       T4207	// R_1st SS ALIGN SIDE BW
OUTP      M12864	// T)R_1st SOL ALIGN SIDE FW >
// ======================== 2nd BENDING ==========================
; L93
LOAD      M13400	// T)R_2nd VC ON/OFF
OUTP      M13320	// T)R_2nd VC ON/OFF PLS
; L94
LOAD      M13320	// T)R_2nd VC ON/OFF PLS
MPUSH
AND NOT   P00146	// R_2nd DIE VACUUM EJECTOR ON
OUTP      M13322	// T)R_2nd VC ON
MPOP
AND       P00146	// R_2nd DIE VACUUM EJECTOR ON
OUTP      M13324	// T)R_2nd VC OFF
; L96
LOAD      M13402	// T)R_2nd SOL CLAMP.L UP/DN
OUTP      M13330	// T)R_2nd SOL CLAMP.L UP/DN PLS
; L97
LOAD      M13330	// T)R_2nd SOL CLAMP.L UP/DN PLS
MPUSH
AND       T4221	// R_2nd SS CLAMP.L DN
OUTP      M13332	// T)R_2nd SOL CLAMP.L UP >
MPOP
AND       T4220	// R_2nd SS CLAMP.L UP
AND       T4223	// R_2nd SS CLAMP.R DN
AND       M04161	// R_2nd_16 T Pos.2nd WORK
OUTP      M13334	// T)R_2nd SOL CLAMP.L DN >
; L99
LOAD      M13404	// T)R_2nd SOL CLAMP.R UP/DN
OUTP      M13340	// T)R_2nd SOL CLAMP.R UP/DN PLS
; L100
LOAD      M13340	// T)R_2nd SOL CLAMP.R UP/DN PLS
MPUSH
AND       T4223	// R_2nd SS CLAMP.R DN
AND       T4220	// R_2nd SS CLAMP.L UP
OUTP      M13342	// T)R_2nd SOL CLAMP.R UP >
MPOP
AND       T4222	// R_2nd SS CLAMP.R UP
AND       F00099
AND       M04161	// R_2nd_16 T Pos.2nd WORK
OUTP      M13344	// T)R_2nd SOL CLAMP.R DN >

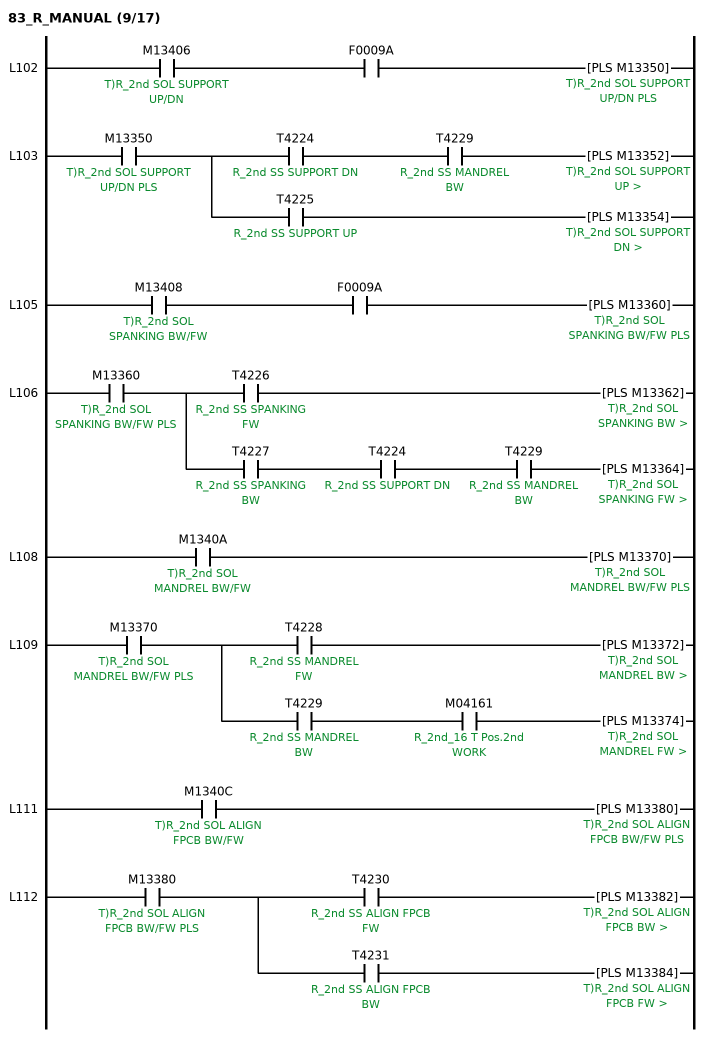
; L102
LOAD      M13406	// T)R_2nd SOL SUPPORT UP/DN
AND       F0009A
OUTP      M13350	// T)R_2nd SOL SUPPORT UP/DN PLS
; L103
LOAD      M13350	// T)R_2nd SOL SUPPORT UP/DN PLS
MPUSH
AND       T4224	// R_2nd SS SUPPORT DN
AND       T4229	// R_2nd SS MANDREL BW
OUTP      M13352	// T)R_2nd SOL SUPPORT UP >
MPOP
AND       T4225	// R_2nd SS SUPPORT UP
OUTP      M13354	// T)R_2nd SOL SUPPORT DN >
; L105
LOAD      M13408	// T)R_2nd SOL SPANKING BW/FW
AND       F0009A
OUTP      M13360	// T)R_2nd SOL SPANKING BW/FW PLS
; L106
LOAD      M13360	// T)R_2nd SOL SPANKING BW/FW PLS
MPUSH
AND       T4226	// R_2nd SS SPANKING FW
OUTP      M13362	// T)R_2nd SOL SPANKING BW >
MPOP
AND       T4227	// R_2nd SS SPANKING BW
AND       T4224	// R_2nd SS SUPPORT DN
AND       T4229	// R_2nd SS MANDREL BW
OUTP      M13364	// T)R_2nd SOL SPANKING FW >
; L108
LOAD      M1340A	// T)R_2nd SOL MANDREL BW/FW
OUTP      M13370	// T)R_2nd SOL MANDREL BW/FW PLS
; L109
LOAD      M13370	// T)R_2nd SOL MANDREL BW/FW PLS
MPUSH
AND       T4228	// R_2nd SS MANDREL FW
OUTP      M13372	// T)R_2nd SOL MANDREL BW >
MPOP
AND       T4229	// R_2nd SS MANDREL BW
AND       M04161	// R_2nd_16 T Pos.2nd WORK
OUTP      M13374	// T)R_2nd SOL MANDREL FW >
; L111
LOAD      M1340C	// T)R_2nd SOL ALIGN FPCB BW/FW
OUTP      M13380	// T)R_2nd SOL ALIGN FPCB BW/FW PLS
; L112
LOAD      M13380	// T)R_2nd SOL ALIGN FPCB BW/FW PLS
MPUSH
AND       T4230	// R_2nd SS ALIGN FPCB FW
OUTP      M13382	// T)R_2nd SOL ALIGN FPCB BW >
MPOP
AND       T4231	// R_2nd SS ALIGN FPCB BW
OUTP      M13384	// T)R_2nd SOL ALIGN FPCB FW >

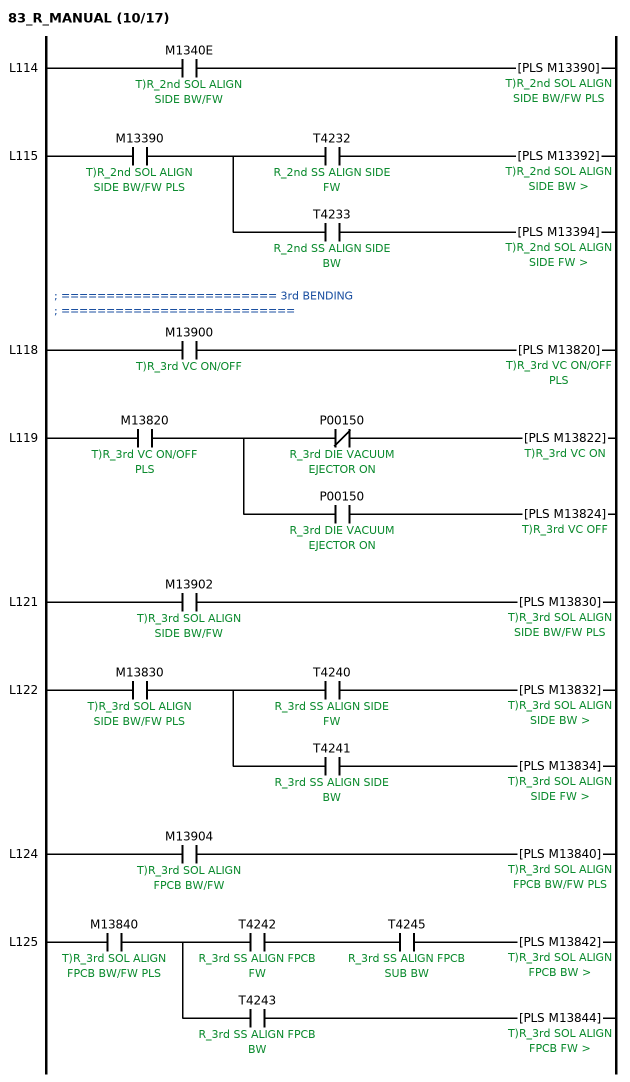
; L114
LOAD      M1340E	// T)R_2nd SOL ALIGN SIDE BW/FW
OUTP      M13390	// T)R_2nd SOL ALIGN SIDE BW/FW PLS
; L115
LOAD      M13390	// T)R_2nd SOL ALIGN SIDE BW/FW PLS
MPUSH
AND       T4232	// R_2nd SS ALIGN SIDE FW
OUTP      M13392	// T)R_2nd SOL ALIGN SIDE BW >
MPOP
AND       T4233	// R_2nd SS ALIGN SIDE BW
OUTP      M13394	// T)R_2nd SOL ALIGN SIDE FW >
// ======================== 3rd BENDING ==========================
; L118
LOAD      M13900	// T)R_3rd VC ON/OFF
OUTP      M13820	// T)R_3rd VC ON/OFF PLS
; L119
LOAD      M13820	// T)R_3rd VC ON/OFF PLS
MPUSH
AND NOT   P00150	// R_3rd DIE VACUUM EJECTOR ON
OUTP      M13822	// T)R_3rd VC ON
MPOP
AND       P00150	// R_3rd DIE VACUUM EJECTOR ON
OUTP      M13824	// T)R_3rd VC OFF
; L121
LOAD      M13902	// T)R_3rd SOL ALIGN SIDE BW/FW
OUTP      M13830	// T)R_3rd SOL ALIGN SIDE BW/FW PLS
; L122
LOAD      M13830	// T)R_3rd SOL ALIGN SIDE BW/FW PLS
MPUSH
AND       T4240	// R_3rd SS ALIGN SIDE FW
OUTP      M13832	// T)R_3rd SOL ALIGN SIDE BW >
MPOP
AND       T4241	// R_3rd SS ALIGN SIDE BW
OUTP      M13834	// T)R_3rd SOL ALIGN SIDE FW >
; L124
LOAD      M13904	// T)R_3rd SOL ALIGN FPCB BW/FW
OUTP      M13840	// T)R_3rd SOL ALIGN FPCB BW/FW PLS
; L125
LOAD      M13840	// T)R_3rd SOL ALIGN FPCB BW/FW PLS
MPUSH
AND       T4242	// R_3rd SS ALIGN FPCB FW
AND       T4245	// R_3rd SS ALIGN FPCB SUB BW
OUTP      M13842	// T)R_3rd SOL ALIGN FPCB BW >
MPOP
AND       T4243	// R_3rd SS ALIGN FPCB BW
OUTP      M13844	// T)R_3rd SOL ALIGN FPCB FW >

